KUKA KRL program: EPS_2_251806_MH01A_A_20260212042228.src

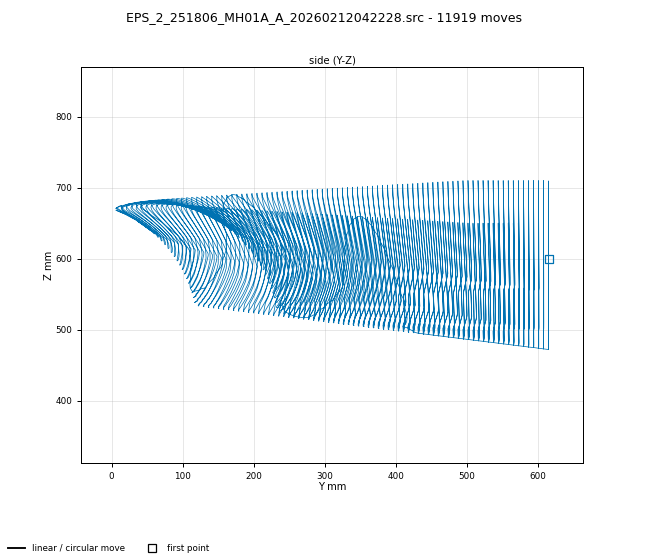
[picture p0: tool path of EPS_2_251806_MH01A_A_20260212042228.src, 11919 of 11921 moves have a stored position in this frame; points joined in program order, loops and branches not executed]
&ACCESS RVP
&REL 4
&COMMENT QRS 19112012
&PARAM EDITMASK = *
DEF PART()
EXT BAS (BAS_COMMAND :IN,REAL :IN )
INT I
BAS (#INITMOV,0 )

;KUKA QRS Post kuka4.cps  Date:22-06-2017 !

File_ID=3008

QRS_PRE_INIT()

;Init var - Until changes are made in qrs_pre_init
Outlet_Square_prg=0
Inlet_1_Square_prg=0
Inlet_2_Square_prg=0
Inlet_3_Square_prg=0
Inlet_4_Square_prg=0
Inlet_5_Square_prg=0

Outlet_1={X 0.000, Y 496.750, Z 561.000, B 0.000, E1 0.000 }
Inlet_1={X 0.000, Y 501.240, Z 501.000, B 0.000, E1 220.000 }
Outlet_1_type=299
Inlet_1_type=299
;QRS#1=Sidecore dimensions
;QRS#2=300-12" PVC SDR 35
;QRS#3=300-12" PVC SDR 35
;QRS#4=
;QRS#5=
;QRS#6=
;QRS#7=
;QRS#8=
;QRS#9=16M PSX
;QRS#10=16M PSX
;QRS#11=
;QRS#12=
;QRS#13=
;QRS#14=
;QRS#15=
;QRS#16=1220x127x991 3,25'
;QRS#17=EPS Height
;QRS#18=710,5
;QRS#19=*
;QRS#20= UPDATED VERSION 22-06-2017
;QRS#21=*
Outlet_Square=0150
Inlet_1_Square=0150
Inlet_2_Square=0
Inlet_3_Square=0
Inlet_4_Square=0
Inlet_5_Square=0
Mill_Square=1
Outlet_Square_Prg=206
Inlet_1_Square_prg=206

QRS_INIT()

$ADVANCE=5

; T1
PTP {E1 173.593,E2 173.593}
PTP {X 0,Y 615.505,A -85,B 0,C 180,E1 173.593,E2 173.593,E3 0,E4 0,E5 0,E6 0}
QRS_SPEED_INIT()
LIN {X 0,Y 615.505,Z 600,A -85,B 0,C 180,E1 173.593,E2 173.593,E3 0,E4 0,E5 0,E6 0} C_VEL
LIN {X 0,Y 615.505,Z 482.498,A -85,B 0,C 180,E1 173.593,E2 173.593} C_VEL
LIN {X 0,Y 615.505,Z 474.321,A -85,B 0,C 180,E1 173.593,E2 173.593} C_VEL
LIN {X 0,Y 615.491,Z 472.321,A -85,B 0,C 180,E1 173.407,E2 173.407} C_VEL
LIN {X 0,Y 615.481,Z 472.326,A -85,B 0,C 180,E1 170.801,E2 170.801} C_VEL
LIN {X 0,Y 615.48,Z 472.325,A -85,B 0,C 180,E1 168.139,E2 168.139} C_VEL
LIN {X 0,Y 615.489,Z 472.322,A -85,B 0,C 180,E1 165.451,E2 165.451} C_VEL
LIN {X 0,Y 615.493,Z 472.323,A -85,B 0,C 180,E1 162.729,E2 162.729} C_VEL
LIN {X 0,Y 615.484,Z 472.323,A -85,B 0,C 180,E1 159.967,E2 159.967} C_VEL
LIN {X 0,Y 615.483,Z 472.325,A -85,B 0,C 180,E1 157.155,E2 157.155} C_VEL
LIN {X 0,Y 615.498,Z 472.322,A -85,B 0,C 180,E1 154.284,E2 154.284} C_VEL
LIN {X 0,Y 615.484,Z 472.323,A -85,B 0,C 180,E1 151.548,E2 151.548} C_VEL
LIN {X 0,Y 615.482,Z 472.324,A -85,B 0,C 180,E1 148.912,E2 148.912} C_VEL
LIN {X 0,Y 615.491,Z 472.325,A -85,B 0,C 180,E1 146.463,E2 146.463} C_VEL
LIN {X 0,Y 615.483,Z 472.322,A -85,B 0,C 180,E1 143.574,E2 143.574} C_VEL
LIN {X 0,Y 615.495,Z 472.325,A -85,B 0,C 180,E1 140.935,E2 140.935} C_VEL
LIN {X 0,Y 615.496,Z 472.323,A -85,B 0,C 180,E1 138.526,E2 138.526} C_VEL
LIN {X 0,Y 615.482,Z 472.323,A -85,B 0,C 180,E1 135.849,E2 135.849} C_VEL
LIN {X 0,Y 615.486,Z 472.326,A -85,B 0,C 180,E1 133.047,E2 133.047} C_VEL
LIN {X 0,Y 615.496,Z 472.322,A -85,B 0,C 180,E1 130.089,E2 130.089} C_VEL
LIN {X 0,Y 615.491,Z 472.321,A -85,B 0,C 180,E1 127.241,E2 127.241} C_VEL
LIN {X 0,Y 615.483,Z 472.323,A -85,B 0,C 180,E1 124.699,E2 124.699} C_VEL
LIN {X 0,Y 615.487,Z 472.325,A -85,B 0,C 180,E1 122.33,E2 122.33} C_VEL
LIN {X 0,Y 615.486,Z 472.325,A -85,B 0,C 180,E1 119.793,E2 119.793} C_VEL
LIN {X 0,Y 615.491,Z 472.321,A -85,B 0,C 180,E1 117.045,E2 117.045} C_VEL
LIN {X 0,Y 615.497,Z 472.322,A -85,B 0,C 180,E1 114.271,E2 114.271} C_VEL
LIN {X 0,Y 615.48,Z 472.325,A -85,B 0,C 180,E1 111.431,E2 111.431} C_VEL
LIN {X 0,Y 615.484,Z 472.323,A -85,B 0,C 180,E1 108.602,E2 108.602} C_VEL
LIN {X 0,Y 615.495,Z 472.321,A -85,B 0,C 180,E1 105.904,E2 105.904} C_VEL
LIN {X 0,Y 615.487,Z 472.324,A -85,B 0,C 180,E1 103.201,E2 103.201} C_VEL
LIN {X 0,Y 615.48,Z 472.324,A -85,B 0,C 180,E1 100.527,E2 100.527} C_VEL
LIN {X 0,Y 615.489,Z 472.326,A -85,B 0,C 180,E1 97.875,E2 97.875} C_VEL
LIN {X 0,Y 615.484,Z 472.322,A -85,B 0,C 180,E1 95.241,E2 95.241} C_VEL
LIN {X 0,Y 615.483,Z 472.325,A -85,B 0,C 180,E1 92.617,E2 92.617} C_VEL
LIN {X 0,Y 615.492,Z 472.323,A -85,B 0,C 180,E1 90,E2 90} C_VEL
LIN {X 0,Y 615.498,Z 472.416,A -85,B 0,C 180,E1 88.037,E2 88.037} C_VEL
LIN {X 0,Y 615.48,Z 475.112,A -85,B 0,C 180,E1 85.415,E2 85.415} C_VEL
LIN {X 0,Y 615.489,Z 477.991,A -85,B 0,C 180,E1 82.784,E2 82.784} C_VEL
LIN {X 0,Y 615.484,Z 480.998,A -85,B 0,C 180,E1 80.138,E2 80.138} C_VEL
LIN {X 0,Y 615.491,Z 484.127,A -85,B 0,C 180,E1 77.47,E2 77.47} C_VEL
LIN {X 0,Y 615.489,Z 487.344,A -85,B 0,C 180,E1 74.774,E2 74.774} C_VEL
LIN {X 0,Y 615.487,Z 490.698,A -85,B 0,C 180,E1 72.043,E2 72.043} C_VEL
LIN {X 0,Y 615.478,Z 494.15,A -85,B 0,C 180,E1 69.269,E2 69.269} C_VEL
LIN {X 0,Y 615.48,Z 496.826,A -85,B 0,C 180,E1 67.155,E2 67.155} C_VEL
LIN {X 0,Y 615.477,Z 498.079,A -85,B 0,C 180,E1 66.288,E2 66.288} C_VEL
LIN {X 0,Y 615.487,Z 512.595,A -85,B 0,C 180,E1 66.049,E2 66.049} C_VEL
LIN {X 0,Y 615.485,Z 527.058,A -85,B 0,C 180,E1 65.683,E2 65.683} C_VEL
LIN {X 0,Y 615.479,Z 541.48,A -85,B 0,C 180,E1 65.188,E2 65.188} C_VEL
LIN {X 0,Y 615.481,Z 555.329,A -85,B 0,C 180,E1 64.578,E2 64.578} C_VEL
LIN {X 0,Y 615.499,Z 568.988,A -85,B 0,C 180,E1 63.83,E2 63.83} C_VEL
LIN {X 0,Y 615.498,Z 582.101,A -85,B 0,C 180,E1 62.954,E2 62.954} C_VEL
LIN {X 0,Y 615.493,Z 592.977,A -85,B 0,C 180,E1 62.085,E2 62.085} C_VEL
LIN {X 0,Y 615.494,Z 602.897,A -85,B 0,C 180,E1 61.156,E2 61.156} C_VEL
LIN {X 0,Y 615.497,Z 613.099,A -85,B 0,C 180,E1 60.023,E2 60.023} C_VEL
LIN {X 0,Y 615.497,Z 622.489,A -85,B 0,C 180,E1 58.765,E2 58.765} C_VEL
LIN {X 0,Y 615.493,Z 629.992,A -85,B 0,C 180,E1 57.543,E2 57.543} C_VEL
LIN {X 0,Y 615.492,Z 636.558,A -85,B 0,C 180,E1 56.223,E2 56.223} C_VEL
LIN {X 0,Y 615.487,Z 640.708,A -85,B 0,C 180,E1 55.185,E2 55.185} C_VEL
LIN {X 0,Y 615.493,Z 643.983,A -85,B 0,C 180,E1 54.166,E2 54.166} C_VEL
LIN {X 0,Y 615.493,Z 647.292,A -85,B 0,C 180,E1 52.759,E2 52.759} C_VEL
LIN {X 0,Y 615.494,Z 648.577,A -85,B 0,C 180,E1 51.932,E2 51.932} C_VEL
LIN {X 0,Y 615.49,Z 649.536,A -85,B 0,C 180,E1 50.938,E2 50.938} C_VEL
LIN {X 0,Y 615.498,Z 649.883,A -85,B 0,C 180,E1 49.91,E2 49.91} C_VEL
LIN {X 0,Y 615.491,Z 649.22,A -85,B 0,C 180,E1 48.527,E2 48.527} C_VEL
LIN {X 0,Y 615.491,Z 646.908,A -85,B 0,C 180,E1 46.953,E2 46.953} C_VEL
LIN {X 0,Y 615.493,Z 643.151,A -85,B 0,C 180,E1 45.461,E2 45.461} C_VEL
LIN {X 0,Y 615.492,Z 638.543,A -85,B 0,C 180,E1 44.15,E2 44.15} C_VEL
LIN {X 0,Y 615.494,Z 631.812,A -85,B 0,C 180,E1 42.7,E2 42.7} C_VEL
LIN {X 0,Y 615.495,Z 624.699,A -85,B 0,C 180,E1 41.474,E2 41.474} C_VEL
LIN {X 0,Y 615.496,Z 615.806,A -85,B 0,C 180,E1 40.22,E2 40.22} C_VEL
LIN {X 0,Y 615.495,Z 605.907,A -85,B 0,C 180,E1 39.064,E2 39.064} C_VEL
LIN {X 0,Y 615.496,Z 595.163,A -85,B 0,C 180,E1 38.014,E2 38.014} C_VEL
LIN {X 0,Y 615.495,Z 582.905,A -85,B 0,C 180,E1 37.014,E2 37.014} C_VEL
LIN {X 0,Y 615.497,Z 569.826,A -85,B 0,C 180,E1 36.13,E2 36.13} C_VEL
LIN {X 0,Y 615.481,Z 556.024,A -85,B 0,C 180,E1 35.366,E2 35.366} C_VEL
LIN {X 0,Y 615.49,Z 542.45,A -85,B 0,C 180,E1 34.759,E2 34.759} C_VEL
LIN {X 0,Y 615.477,Z 527.351,A -85,B 0,C 180,E1 34.235,E2 34.235} C_VEL
LIN {X 0,Y 615.487,Z 513.002,A -85,B 0,C 180,E1 33.87,E2 33.87} C_VEL
LIN {X 0,Y 615.491,Z 497.929,A -85,B 0,C 180,E1 33.611,E2 33.611} C_VEL
LIN {X 0,Y 615.483,Z 494.501,A -85,B 0,C 180,E1 30.92,E2 30.92} C_VEL
LIN {X 0,Y 615.483,Z 491.414,A -85,B 0,C 180,E1 28.451,E2 28.451} C_VEL
LIN {X 0,Y 615.493,Z 487.874,A -85,B 0,C 180,E1 25.571,E2 25.571} C_VEL
LIN {X 0,Y 615.482,Z 484.601,A -85,B 0,C 180,E1 22.845,E2 22.845} C_VEL
LIN {X 0,Y 615.477,Z 481.304,A -85,B 0,C 180,E1 20.033,E2 20.033} C_VEL
LIN {X 0,Y 615.492,Z 478.15,A -85,B 0,C 180,E1 17.271,E2 17.271} C_VEL
LIN {X 0,Y 615.487,Z 475.186,A -85,B 0,C 180,E1 14.549,E2 14.549} C_VEL
LIN {X 0,Y 615.485,Z 472.509,A -85,B 0,C 180,E1 11.861,E2 11.861} C_VEL
LIN {X 0,Y 615.479,Z 472.312,A -85,B 0,C 180,E1 9.199,E2 9.199} C_VEL
LIN {X 0,Y 615.491,Z 472.313,A -85,B 0,C 180,E1 6.557,E2 6.557} C_VEL
LIN {X 0,Y 615.488,Z 472.319,A -85,B 0,C 180,E1 3.929,E2 3.929} C_VEL
LIN {X 0,Y 615.485,Z 472.309,A -85,B 0,C 180,E1 1.309,E2 1.309} C_VEL
LIN {X 0,Y 615.485,Z 472.321,A -85,B 0,C 180,E1 -1.308,E2 -1.308} C_VEL
LIN {X 0,Y 615.475,Z 472.316,A -85,B 0,C 180,E1 -3.928,E2 -3.928} C_VEL
LIN {X 0,Y 615.492,Z 472.31,A -85,B 0,C 180,E1 -6.588,E2 -6.588} C_VEL
LIN {X 0,Y 615.487,Z 472.325,A -85,B 0,C 180,E1 -9.199,E2 -9.199} C_VEL
LIN {X 0,Y 615.479,Z 472.311,A -85,B 0,C 180,E1 -11.861,E2 -11.861} C_VEL
LIN {X 0,Y 615.491,Z 472.318,A -85,B 0,C 180,E1 -14.549,E2 -14.549} C_VEL
LIN {X 0,Y 615.48,Z 472.314,A -85,B 0,C 180,E1 -17.271,E2 -17.271} C_VEL
LIN {X 0,Y 615.479,Z 472.316,A -85,B 0,C 180,E1 -20.033,E2 -20.033} C_VEL
LIN {X 0,Y 615.482,Z 472.316,A -85,B 0,C 180,E1 -22.845,E2 -22.845} C_VEL
LIN {X 0,Y 615.493,Z 472.312,A -85,B 0,C 180,E1 -25.715,E2 -25.715} C_VEL
LIN {X 0,Y 615.489,Z 472.312,A -85,B 0,C 180,E1 -28.658,E2 -28.658} C_VEL
LIN {X 0,Y 615.477,Z 472.312,A -85,B 0,C 180,E1 -31.085,E2 -31.085} C_VEL
LIN {X 0,Y 615.485,Z 472.319,A -85,B 0,C 180,E1 -33.535,E2 -33.535} C_VEL
LIN {X 0,Y 615.486,Z 472.323,A -85,B 0,C 180,E1 -35.834,E2 -35.834} C_VEL
LIN {X 0,Y 615.478,Z 472.316,A -85,B 0,C 180,E1 -38.069,E2 -38.069} C_VEL
LIN {X 0,Y 615.484,Z 472.31,A -85,B 0,C 180,E1 -40.607,E2 -40.607} C_VEL
LIN {X 0,Y 615.497,Z 472.324,A -85,B 0,C 180,E1 -43.244,E2 -43.244} C_VEL
LIN {X 0,Y 615.482,Z 472.31,A -85,B 0,C 180,E1 -46.003,E2 -46.003} C_VEL
LIN {X 0,Y 615.492,Z 472.352,A -85,B 0,C 180,E1 -48.716,E2 -48.716} C_VEL
LIN {X 0,Y 615.483,Z 479.207,A -85,B 0,C 180,E1 -51.096,E2 -51.096} C_VEL
LIN {X 0,Y 615.486,Z 486.794,A -85,B 0,C 180,E1 -53.576,E2 -53.576} C_VEL
LIN {X 0,Y 615.496,Z 495.763,A -85,B 0,C 180,E1 -56.465,E2 -56.465} C_VEL
LIN {X 0,Y 615.478,Z 504.122,A -85,B 0,C 180,E1 -59.08,E2 -59.08} C_VEL
LIN {X 0,Y 615.481,Z 512.228,A -85,B 0,C 180,E1 -61.551,E2 -61.551} C_VEL
LIN {X 0,Y 615.493,Z 521.4,A -85,B 0,C 180,E1 -64.285,E2 -64.285} C_VEL
LIN {X 0,Y 615.48,Z 531.274,A -85,B 0,C 180,E1 -67.155,E2 -67.155} C_VEL
LIN {X 0,Y 615.492,Z 541.126,A -85,B 0,C 180,E1 -69.967,E2 -69.967} C_VEL
LIN {X 0,Y 615.485,Z 550.985,A -85,B 0,C 180,E1 -72.729,E2 -72.729} C_VEL
LIN {X 0,Y 615.489,Z 554.183,A -85,B 0,C 180,E1 -73.618,E2 -73.618} C_VEL
LIN {X 0,Y 615.495,Z 570.381,A -85,B 0,C 180,E1 -73.865,E2 -73.865} C_VEL
LIN {X 0,Y 615.48,Z 585.284,A -85,B 0,C 180,E1 -74.222,E2 -74.222} C_VEL
LIN {X 0,Y 615.484,Z 599.424,A -85,B 0,C 180,E1 -74.689,E2 -74.689} C_VEL
LIN {X 0,Y 615.485,Z 613.357,A -85,B 0,C 180,E1 -75.282,E2 -75.282} C_VEL
LIN {X 0,Y 615.499,Z 626.673,A -85,B 0,C 180,E1 -75.986,E2 -75.986} C_VEL
LIN {X 0,Y 615.498,Z 639.314,A -85,B 0,C 180,E1 -76.799,E2 -76.799} C_VEL
LIN {X 0,Y 615.496,Z 650.292,A -85,B 0,C 180,E1 -77.637,E2 -77.637} C_VEL
LIN {X 0,Y 615.497,Z 661.353,A -85,B 0,C 180,E1 -78.64,E2 -78.64} C_VEL
LIN {X 0,Y 615.496,Z 672.068,A -85,B 0,C 180,E1 -79.806,E2 -79.806} C_VEL
LIN {X 0,Y 615.497,Z 680.987,A -85,B 0,C 180,E1 -80.967,E2 -80.967} C_VEL
LIN {X 0,Y 615.494,Z 688.391,A -85,B 0,C 180,E1 -82.124,E2 -82.124} C_VEL
LIN {X 0,Y 615.49,Z 695.271,A -85,B 0,C 180,E1 -83.443,E2 -83.443} C_VEL
LIN {X 0,Y 615.491,Z 700.665,A -85,B 0,C 180,E1 -84.759,E2 -84.759} C_VEL
LIN {X 0,Y 615.495,Z 704.739,A -85,B 0,C 180,E1 -86.071,E2 -86.071} C_VEL
LIN {X 0,Y 615.495,Z 707.599,A -85,B 0,C 180,E1 -87.382,E2 -87.382} C_VEL
LIN {X 0,Y 615.493,Z 709.306,A -85,B 0,C 180,E1 -88.691,E2 -88.691} C_VEL
LIN {X 0,Y 615.491,Z 709.889,A -85,B 0,C 180,E1 -90,E2 -90} C_VEL
LIN {X 0,Y 615.493,Z 709.307,A -85,B 0,C 180,E1 -91.308,E2 -91.308} C_VEL
LIN {X 0,Y 615.495,Z 707.6,A -85,B 0,C 180,E1 -92.617,E2 -92.617} C_VEL
LIN {X 0,Y 615.495,Z 704.741,A -85,B 0,C 180,E1 -93.928,E2 -93.928} C_VEL
LIN {X 0,Y 615.491,Z 700.668,A -85,B 0,C 180,E1 -95.241,E2 -95.241} C_VEL
LIN {X 0,Y 615.49,Z 695.155,A -85,B 0,C 180,E1 -96.581,E2 -96.581} C_VEL
LIN {X 0,Y 615.494,Z 688.396,A -85,B 0,C 180,E1 -97.875,E2 -97.875} C_VEL
LIN {X 0,Y 615.497,Z 679.812,A -85,B 0,C 180,E1 -99.198,E2 -99.198} C_VEL
LIN {X 0,Y 615.494,Z 670.672,A -85,B 0,C 180,E1 -100.36,E2 -100.36} C_VEL
LIN {X 0,Y 615.497,Z 661.359,A -85,B 0,C 180,E1 -101.359,E2 -101.359} C_VEL
LIN {X 0,Y 615.496,Z 650.3,A -85,B 0,C 180,E1 -102.362,E2 -102.362} C_VEL
LIN {X 0,Y 615.498,Z 638.161,A -85,B 0,C 180,E1 -103.284,E2 -103.284} C_VEL
LIN {X 0,Y 615.498,Z 625.407,A -85,B 0,C 180,E1 -104.089,E2 -104.089} C_VEL
LIN {X 0,Y 615.486,Z 611.623,A -85,B 0,C 180,E1 -104.802,E2 -104.802} C_VEL
LIN {X 0,Y 615.48,Z 597.199,A -85,B 0,C 180,E1 -105.395,E2 -105.395} C_VEL
LIN {X 0,Y 615.484,Z 582.272,A -85,B 0,C 180,E1 -105.862,E2 -105.862} C_VEL
LIN {X 0,Y 615.496,Z 566.874,A -85,B 0,C 180,E1 -106.2,E2 -106.2} C_VEL
LIN {X 0,Y 615.489,Z 554.125,A -85,B 0,C 180,E1 -106.398,E2 -106.398} C_VEL
LIN {X 0,Y 615.485,Z 544.833,A -85,B 0,C 180,E1 -108.991,E2 -108.991} C_VEL
LIN {X 0,Y 615.486,Z 534.967,A -85,B 0,C 180,E1 -111.783,E2 -111.783} C_VEL
LIN {X 0,Y 615.487,Z 526.34,A -85,B 0,C 180,E1 -114.271,E2 -114.271} C_VEL
LIN {X 0,Y 615.491,Z 516.906,A -85,B 0,C 180,E1 -117.046,E2 -117.046} C_VEL
LIN {X 0,Y 615.485,Z 507.787,A -85,B 0,C 180,E1 -119.794,E2 -119.794} C_VEL
LIN {X 0,Y 615.481,Z 499.186,A -85,B 0,C 180,E1 -122.457,E2 -122.457} C_VEL
LIN {X 0,Y 615.496,Z 490.532,A -85,B 0,C 180,E1 -125.213,E2 -125.213} C_VEL
LIN {X 0,Y 615.489,Z 481.785,A -85,B 0,C 180,E1 -128.067,E2 -128.067} C_VEL
LIN {X 0,Y 615.477,Z 474.341,A -85,B 0,C 180,E1 -130.606,E2 -130.606} C_VEL
LIN {X 0,Y 615.49,Z 472.322,A -85,B 0,C 180,E1 -131.378,E2 -131.378} C_VEL
LIN {X 0,Y 615.492,Z 472.323,A -85,B 0,C 180,E1 -134.148,E2 -134.148} C_VEL
LIN {X 0,Y 615.488,Z 472.322,A -85,B 0,C 180,E1 -136.951,E2 -136.951} C_VEL
LIN {X 0,Y 615.495,Z 472.325,A -85,B 0,C 180,E1 -139.908,E2 -139.908} C_VEL
LIN {X 0,Y 615.481,Z 472.324,A -85,B 0,C 180,E1 -142.758,E2 -142.758} C_VEL
LIN {X 0,Y 615.491,Z 472.326,A -85,B 0,C 180,E1 -145.297,E2 -145.297} C_VEL
LIN {X 0,Y 615.49,Z 472.325,A -85,B 0,C 180,E1 -147.667,E2 -147.667} C_VEL
LIN {X 0,Y 615.488,Z 472.322,A -85,B 0,C 180,E1 -150.203,E2 -150.203} C_VEL
LIN {X 0,Y 615.492,Z 472.325,A -85,B 0,C 180,E1 -152.951,E2 -152.951} C_VEL
LIN {X 0,Y 615.479,Z 472.323,A -85,B 0,C 180,E1 -155.728,E2 -155.728} C_VEL
LIN {X 0,Y 615.499,Z 472.325,A -85,B 0,C 180,E1 -158.569,E2 -158.569} C_VEL
LIN {X 0,Y 615.495,Z 472.32,A -85,B 0,C 180,E1 -161.389,E2 -161.389} C_VEL
LIN {X 0,Y 615.491,Z 472.326,A -85,B 0,C 180,E1 -164.095,E2 -164.095} C_VEL
LIN {X 0,Y 615.48,Z 472.323,A -85,B 0,C 180,E1 -166.799,E2 -166.799} C_VEL
LIN {X 0,Y 615.495,Z 472.324,A -85,B 0,C 180,E1 -169.473,E2 -169.473} C_VEL
LIN {X 0,Y 615.483,Z 472.323,A -85,B 0,C 180,E1 -172.125,E2 -172.125} C_VEL
LIN {X 0,Y 615.487,Z 472.323,A -85,B 0,C 180,E1 -174.759,E2 -174.759} C_VEL
LIN {X 0,Y 615.496,Z 472.324,A -85,B 0,C 180,E1 -177.382,E2 -177.382} C_VEL
LIN {X 0,Y 615.477,Z 472.324,A -85,B 0,C 180,E1 -180,E2 -180} C_VEL
LIN {X 0,Y 615.494,Z 472.323,A -85,B 0,C 180,E1 -182.618,E2 -182.618} C_VEL
LIN {X 0,Y 615.491,Z 472.323,A -85,B 0,C 180,E1 -185.241,E2 -185.241} C_VEL
LIN {X 0,Y 615.491,Z 472.321,A -85,B 0,C 180,E1 -186.593,E2 -186.593} C_VEL
LIN {X 0,Y 614.815,Z 472.47,A -85,B 0,C 180,E1 -187.139,E2 -187.139} C_VEL
LIN {X 0,Y 611.975,Z 472.882,A -85,B 0,C 180,E1 -188.025,E2 -188.025} C_VEL
LIN {X 0,Y 609.579,Z 473.194,A -85,B 0,C 180,E1 -188.737,E2 -188.737} C_VEL
LIN {X 0,Y 608.542,Z 473.312,A -85,B 0,C 180,E1 -189.287,E2 -189.287} C_VEL
LIN {X 0,Y 608.453,Z 473.321,A -85,B 0,C 180,E1 -189.473,E2 -189.473} C_VEL
LIN {X 0,Y 608.457,Z 473.32,A -85,B 0,C 180,E1 -192,E2 -192} C_VEL
LIN {X 0,Y 608.476,Z 473.319,A -85,B 0,C 180,E1 -194.721,E2 -194.721} C_VEL
LIN {X 0,Y 608.457,Z 473.32,A -85,B 0,C 180,E1 -197.477,E2 -197.477} C_VEL
LIN {X 0,Y 608.462,Z 473.321,A -85,B 0,C 180,E1 -200.275,E2 -200.275} C_VEL
LIN {X 0,Y 608.449,Z 473.322,A -85,B 0,C 180,E1 -202.477,E2 -202.477} C_VEL
LIN {X 0,Y 608.453,Z 473.32,A -85,B 0,C 180,E1 -205.301,E2 -205.301} C_VEL
LIN {X 0,Y 608.454,Z 473.32,A -85,B 0,C 180,E1 -207.518,E2 -207.518} C_VEL
LIN {X 0,Y 608.471,Z 473.318,A -85,B 0,C 180,E1 -209.975,E2 -209.975} C_VEL
LIN {X 0,Y 608.465,Z 473.322,A -85,B 0,C 180,E1 -212.525,E2 -212.525} C_VEL
LIN {X 0,Y 608.449,Z 473.32,A -85,B 0,C 180,E1 -215.278,E2 -215.278} C_VEL
LIN {X 0,Y 608.471,Z 473.319,A -85,B 0,C 180,E1 -217.747,E2 -217.747} C_VEL
LIN {X 0,Y 608.477,Z 473.319,A -85,B 0,C 180,E1 -220.334,E2 -220.334} C_VEL
LIN {X 0,Y 608.471,Z 473.319,A -85,B 0,C 180,E1 -223.31,E2 -223.31} C_VEL
LIN {X 0,Y 608.469,Z 473.318,A -85,B 0,C 180,E1 -226.132,E2 -226.132} C_VEL
LIN {X 0,Y 608.461,Z 473.32,A -85,B 0,C 180,E1 -228.825,E2 -228.825} C_VEL
LIN {X 0,Y 608.473,Z 473.317,A -85,B 0,C 180,E1 -231.76,E2 -231.76} C_VEL
LIN {X 0,Y 608.478,Z 473.317,A -85,B 0,C 180,E1 -233.951,E2 -233.951} C_VEL
LIN {X 0,Y 608.463,Z 473.319,A -85,B 0,C 180,E1 -236.33,E2 -236.33} C_VEL
LIN {X 0,Y 608.479,Z 473.318,A -85,B 0,C 180,E1 -238.728,E2 -238.728} C_VEL
LIN {X 0,Y 608.477,Z 473.318,A -85,B 0,C 180,E1 -241.38,E2 -241.38} C_VEL
LIN {X 0,Y 608.479,Z 473.318,A -85,B 0,C 180,E1 -244.279,E2 -244.279} C_VEL
LIN {X 0,Y 608.45,Z 473.321,A -85,B 0,C 180,E1 -246.877,E2 -246.877} C_VEL
LIN {X 0,Y 608.461,Z 473.319,A -85,B 0,C 180,E1 -249.324,E2 -249.324} C_VEL
LIN {X 0,Y 608.455,Z 473.32,A -85,B 0,C 180,E1 -251.829,E2 -251.829} C_VEL
LIN {X 0,Y 608.476,Z 473.318,A -85,B 0,C 180,E1 -254.595,E2 -254.595} C_VEL
LIN {X 0,Y 608.473,Z 473.318,A -85,B 0,C 180,E1 -257.324,E2 -257.324} C_VEL
LIN {X 0,Y 608.454,Z 473.321,A -85,B 0,C 180,E1 -260.023,E2 -260.023} C_VEL
LIN {X 0,Y 608.467,Z 473.318,A -85,B 0,C 180,E1 -262.701,E2 -262.701} C_VEL
LIN {X 0,Y 608.463,Z 473.322,A -85,B 0,C 180,E1 -265.363,E2 -265.363} C_VEL
LIN {X 0,Y 608.466,Z 473.318,A -85,B 0,C 180,E1 -268.015,E2 -268.015} C_VEL
LIN {X 0,Y 608.481,Z 473.318,A -85,B 0,C 180,E1 -270.662,E2 -270.662} C_VEL
LIN {X 0,Y 608.465,Z 473.322,A -85,B 0,C 180,E1 -271.986,E2 -271.986} C_VEL
LIN {X 0,Y 608.449,Z 476,A -85,B 0,C 180,E1 -274.638,E2 -274.638} C_VEL
LIN {X 0,Y 608.453,Z 478.867,A -85,B 0,C 180,E1 -277.3,E2 -277.3} C_VEL
LIN {X 0,Y 608.421,Z 481.906,A -85,B 0,C 180,E1 -279.978,E2 -279.978} C_VEL
LIN {X 0,Y 608.423,Z 485.051,A -85,B 0,C 180,E1 -282.678,E2 -282.678} C_VEL
LIN {X 0,Y 608.419,Z 488.309,A -85,B 0,C 180,E1 -285.407,E2 -285.407} C_VEL
LIN {X 0,Y 608.411,Z 491.684,A -85,B 0,C 180,E1 -288.173,E2 -288.173} C_VEL
LIN {X 0,Y 608.413,Z 495.181,A -85,B 0,C 180,E1 -290.983,E2 -290.983} C_VEL
LIN {X 0,Y 608.429,Z 498.373,A -85,B 0,C 180,E1 -293.508,E2 -293.508} C_VEL
LIN {X 0,Y 608.664,Z 502.587,A -85,B 0,C 180,E1 -293.588,E2 -293.588} C_VEL
LIN {X 0,Y 608.664,Z 517.473,A -85,B 0,C 180,E1 -293.879,E2 -293.879} C_VEL
LIN {X 0,Y 608.622,Z 532.678,A -85,B 0,C 180,E1 -294.315,E2 -294.315} C_VEL
LIN {X 0,Y 608.612,Z 547.393,A -85,B 0,C 180,E1 -294.883,E2 -294.883} C_VEL
LIN {X 0,Y 608.566,Z 561.722,A -85,B 0,C 180,E1 -295.586,E2 -295.586} C_VEL
LIN {X 0,Y 608.539,Z 575.136,A -85,B 0,C 180,E1 -296.4,E2 -296.4} C_VEL
LIN {X 0,Y 608.528,Z 587.703,A -85,B 0,C 180,E1 -297.323,E2 -297.323} C_VEL
LIN {X 0,Y 608.485,Z 598.497,A -85,B 0,C 180,E1 -298.265,E2 -298.265} C_VEL
LIN {X 0,Y 608.484,Z 609.409,A -85,B 0,C 180,E1 -299.398,E2 -299.398} C_VEL
LIN {X 0,Y 608.454,Z 618.664,A -85,B 0,C 180,E1 -300.545,E2 -300.545} C_VEL
LIN {X 0,Y 608.46,Z 626.494,A -85,B 0,C 180,E1 -301.705,E2 -301.705} C_VEL
LIN {X 0,Y 608.442,Z 633.124,A -85,B 0,C 180,E1 -302.88,E2 -302.88} C_VEL
LIN {X 0,Y 608.44,Z 638.578,A -85,B 0,C 180,E1 -304.071,E2 -304.071} C_VEL
LIN {X 0,Y 608.424,Z 642.973,A -85,B 0,C 180,E1 -305.279,E2 -305.279} C_VEL
LIN {X 0,Y 608.422,Z 645.348,A -85,B 0,C 180,E1 -306.094,E2 -306.094} C_VEL
LIN {X 0,Y 608.431,Z 647.777,A -85,B 0,C 180,E1 -307.153,E2 -307.153} C_VEL
LIN {X 0,Y 608.413,Z 649.814,A -85,B 0,C 180,E1 -308.592,E2 -308.592} C_VEL
LIN {X 0,Y 608.412,Z 650.365,A -85,B 0,C 180,E1 -309.444,E2 -309.444} C_VEL
LIN {X 0,Y 608.433,Z 650.44,A -85,B 0,C 180,E1 -310.326,E2 -310.326} C_VEL
LIN {X 0,Y 608.415,Z 649.935,A -85,B 0,C 180,E1 -311.337,E2 -311.337} C_VEL
LIN {X 0,Y 608.437,Z 648.787,A -85,B 0,C 180,E1 -312.331,E2 -312.331} C_VEL
LIN {X 0,Y 608.436,Z 646.996,A -85,B 0,C 180,E1 -313.305,E2 -313.305} C_VEL
LIN {X 0,Y 608.423,Z 643.014,A -85,B 0,C 180,E1 -314.798,E2 -314.798} C_VEL
LIN {X 0,Y 608.429,Z 638.119,A -85,B 0,C 180,E1 -316.126,E2 -316.126} C_VEL
LIN {X 0,Y 608.44,Z 632.234,A -85,B 0,C 180,E1 -317.38,E2 -317.38} C_VEL
LIN {X 0,Y 608.443,Z 624.802,A -85,B 0,C 180,E1 -318.659,E2 -318.659} C_VEL
LIN {X 0,Y 608.474,Z 615.89,A -85,B 0,C 180,E1 -319.914,E2 -319.914} C_VEL
LIN {X 0,Y 608.494,Z 606.137,A -85,B 0,C 180,E1 -321.058,E2 -321.058} C_VEL
LIN {X 0,Y 608.497,Z 595.228,A -85,B 0,C 180,E1 -322.13,E2 -322.13} C_VEL
LIN {X 0,Y 608.518,Z 583.622,A -85,B 0,C 180,E1 -323.089,E2 -323.089} C_VEL
LIN {X 0,Y 608.548,Z 571.35,A -85,B 0,C 180,E1 -323.941,E2 -323.941} C_VEL
LIN {X 0,Y 608.576,Z 557.516,A -85,B 0,C 180,E1 -324.731,E2 -324.731} C_VEL
LIN {X 0,Y 608.624,Z 543.685,A -85,B 0,C 180,E1 -325.368,E2 -325.368} C_VEL
LIN {X 0,Y 608.633,Z 528.133,A -85,B 0,C 180,E1 -325.924,E2 -325.924} C_VEL
LIN {X 0,Y 608.675,Z 512.3,A -85,B 0,C 180,E1 -326.329,E2 -326.329} C_VEL
LIN {X 0,Y 608.519,Z 499.111,A -85,B 0,C 180,E1 -326.556,E2 -326.556} C_VEL
LIN {X 0,Y 608.415,Z 498.384,A -85,B 0,C 180,E1 -326.574,E2 -326.574} C_VEL
LIN {X 0,Y 608.422,Z 494.748,A -85,B 0,C 180,E1 -329.452,E2 -329.452} C_VEL
LIN {X 0,Y 608.431,Z 491.912,A -85,B 0,C 180,E1 -331.732,E2 -331.732} C_VEL
LIN {X 0,Y 608.43,Z 488.29,A -85,B 0,C 180,E1 -334.698,E2 -334.698} C_VEL
LIN {X 0,Y 608.428,Z 484.838,A -85,B 0,C 180,E1 -337.593,E2 -337.593} C_VEL
LIN {X 0,Y 608.43,Z 481.542,A -85,B 0,C 180,E1 -340.428,E2 -340.428} C_VEL
LIN {X 0,Y 608.447,Z 478.394,A -85,B 0,C 180,E1 -343.215,E2 -343.215} C_VEL
LIN {X 0,Y 608.454,Z 475.497,A -85,B 0,C 180,E1 -345.986,E2 -345.986} C_VEL
LIN {X 0,Y 608.445,Z 473.518,A -85,B 0,C 180,E1 -348,E2 -348} C_VEL
LIN {X 0,Y 608.465,Z 473.32,A -85,B 0,C 180,E1 -350.023,E2 -350.023} C_VEL
LIN {X 0,Y 608.46,Z 473.313,A -85,B 0,C 180,E1 -352.7,E2 -352.7} C_VEL
LIN {X 0,Y 608.462,Z 473.315,A -85,B 0,C 180,E1 -355.362,E2 -355.362} C_VEL
LIN {X 0,Y 608.457,Z 473.318,A -85,B 0,C 180,E1 -358.014,E2 -358.014} C_VEL
LIN {X 0,Y 608.479,Z 473.31,A -85,B 0,C 180,E1 -360.662,E2 -360.662} C_VEL
LIN {X 0,Y 608.476,Z 473.318,A -85,B 0,C 180,E1 -363.31,E2 -363.31} C_VEL
LIN {X 0,Y 608.454,Z 473.314,A -85,B 0,C 180,E1 -365.967,E2 -365.967} C_VEL
LIN {X 0,Y 608.46,Z 473.315,A -85,B 0,C 180,E1 -368.636,E2 -368.636} C_VEL
LIN {X 0,Y 608.471,Z 473.316,A -85,B 0,C 180,E1 -371.324,E2 -371.324} C_VEL
LIN {X 0,Y 608.463,Z 473.312,A -85,B 0,C 180,E1 -374.037,E2 -374.037} C_VEL
LIN {X 0,Y 608.475,Z 473.319,A -85,B 0,C 180,E1 -376.783,E2 -376.783} C_VEL
LIN {X 0,Y 608.447,Z 473.314,A -85,B 0,C 180,E1 -379.571,E2 -379.571} C_VEL
LIN {X 0,Y 608.471,Z 473.321,A -85,B 0,C 180,E1 -382.405,E2 -382.405} C_VEL
LIN {X 0,Y 608.451,Z 473.319,A -85,B 0,C 180,E1 -384.571,E2 -384.571} C_VEL
LIN {X 0,Y 608.471,Z 473.311,A -85,B 0,C 180,E1 -387.207,E2 -387.207} C_VEL
LIN {X 0,Y 608.47,Z 473.321,A -85,B 0,C 180,E1 -389.973,E2 -389.973} C_VEL
LIN {X 0,Y 608.462,Z 473.313,A -85,B 0,C 180,E1 -392.523,E2 -392.523} C_VEL
LIN {X 0,Y 608.449,Z 473.317,A -85,B 0,C 180,E1 -395.277,E2 -395.277} C_VEL
LIN {X 0,Y 608.464,Z 473.319,A -85,B 0,C 180,E1 -397.746,E2 -397.746} C_VEL
LIN {X 0,Y 608.446,Z 473.314,A -85,B 0,C 180,E1 -400.329,E2 -400.329} C_VEL
LIN {X 0,Y 608.482,Z 473.32,A -85,B 0,C 180,E1 -403.311,E2 -403.311} C_VEL
LIN {X 0,Y 608.469,Z 473.312,A -85,B 0,C 180,E1 -406.131,E2 -406.131} C_VEL
LIN {X 0,Y 608.476,Z 473.373,A -85,B 0,C 180,E1 -408.522,E2 -408.522} C_VEL
LIN {X 0,Y 608.543,Z 479.468,A -85,B 0,C 180,E1 -410.694,E2 -410.694} C_VEL
LIN {X 0,Y 608.518,Z 487.918,A -85,B 0,C 180,E1 -413.503,E2 -413.503} C_VEL
LIN {X 0,Y 608.525,Z 495.494,A -85,B 0,C 180,E1 -415.934,E2 -415.934} C_VEL
LIN {X 0,Y 608.521,Z 504.27,A -85,B 0,C 180,E1 -418.721,E2 -418.721} C_VEL
LIN {X 0,Y 608.493,Z 512.881,A -85,B 0,C 180,E1 -421.376,E2 -421.376} C_VEL
LIN {X 0,Y 608.496,Z 522.524,A -85,B 0,C 180,E1 -424.274,E2 -424.274} C_VEL
LIN {X 0,Y 608.461,Z 531.392,A -85,B 0,C 180,E1 -426.877,E2 -426.877} C_VEL
LIN {X 0,Y 608.46,Z 539.883,A -85,B 0,C 180,E1 -429.323,E2 -429.323} C_VEL
LIN {X 0,Y 608.442,Z 549.959,A -85,B 0,C 180,E1 -432.176,E2 -432.176} C_VEL
LIN {X 0,Y 608.459,Z 554.427,A -85,B 0,C 180,E1 -433.427,E2 -433.427} C_VEL
LIN {X 0,Y 608.687,Z 568.619,A -85,B 0,C 180,E1 -433.646,E2 -433.646} C_VEL
LIN {X 0,Y 608.634,Z 583.766,A -85,B 0,C 180,E1 -433.997,E2 -433.997} C_VEL
LIN {X 0,Y 608.625,Z 598.304,A -85,B 0,C 180,E1 -434.469,E2 -434.469} C_VEL
LIN {X 0,Y 608.591,Z 611.613,A -85,B 0,C 180,E1 -435.026,E2 -435.026} C_VEL
LIN {X 0,Y 608.569,Z 624.788,A -85,B 0,C 180,E1 -435.709,E2 -435.709} C_VEL
LIN {X 0,Y 608.548,Z 638.199,A -85,B 0,C 180,E1 -436.56,E2 -436.56} C_VEL
LIN {X 0,Y 608.504,Z 650.387,A -85,B 0,C 180,E1 -437.493,E2 -437.493} C_VEL
LIN {X 0,Y 608.497,Z 661.508,A -85,B 0,C 180,E1 -438.508,E2 -438.508} C_VEL
LIN {X 0,Y 608.476,Z 672.297,A -85,B 0,C 180,E1 -439.687,E2 -439.687} C_VEL
LIN {X 0,Y 608.47,Z 681.289,A -85,B 0,C 180,E1 -440.862,E2 -440.862} C_VEL
LIN {X 0,Y 608.458,Z 688.751,A -85,B 0,C 180,E1 -442.033,E2 -442.033} C_VEL
LIN {X 0,Y 608.44,Z 695.86,A -85,B 0,C 180,E1 -443.399,E2 -443.399} C_VEL
LIN {X 0,Y 608.437,Z 701.16,A -85,B 0,C 180,E1 -444.698,E2 -444.698} C_VEL
LIN {X 0,Y 608.431,Z 705.287,A -85,B 0,C 180,E1 -446.026,E2 -446.026} C_VEL
LIN {X 0,Y 608.423,Z 708.184,A -85,B 0,C 180,E1 -447.351,E2 -447.351} C_VEL
LIN {X 0,Y 608.445,Z 709.912,A -85,B 0,C 180,E1 -448.676,E2 -448.676} C_VEL
LIN {X 0,Y 608.431,Z 710.5,A -85,B 0,C 180,E1 -450,E2 -450} C_VEL
LIN {X 0,Y 608.445,Z 709.912,A -85,B 0,C 180,E1 -451.323,E2 -451.323} C_VEL
LIN {X 0,Y 608.423,Z 708.185,A -85,B 0,C 180,E1 -452.648,E2 -452.648} C_VEL
LIN {X 0,Y 608.431,Z 705.289,A -85,B 0,C 180,E1 -453.974,E2 -453.974} C_VEL
LIN {X 0,Y 608.437,Z 701.163,A -85,B 0,C 180,E1 -455.302,E2 -455.302} C_VEL
LIN {X 0,Y 608.436,Z 695.705,A -85,B 0,C 180,E1 -456.633,E2 -456.633} C_VEL
LIN {X 0,Y 608.457,Z 688.755,A -85,B 0,C 180,E1 -457.967,E2 -457.967} C_VEL
LIN {X 0,Y 608.47,Z 681.293,A -85,B 0,C 180,E1 -459.138,E2 -459.138} C_VEL
LIN {X 0,Y 608.476,Z 672.303,A -85,B 0,C 180,E1 -460.313,E2 -460.313} C_VEL
LIN {X 0,Y 608.496,Z 661.515,A -85,B 0,C 180,E1 -461.492,E2 -461.492} C_VEL
LIN {X 0,Y 608.504,Z 650.396,A -85,B 0,C 180,E1 -462.506,E2 -462.506} C_VEL
LIN {X 0,Y 608.548,Z 638.209,A -85,B 0,C 180,E1 -463.439,E2 -463.439} C_VEL
LIN {X 0,Y 608.575,Z 625.232,A -85,B 0,C 180,E1 -464.265,E2 -464.265} C_VEL
LIN {X 0,Y 608.59,Z 611.626,A -85,B 0,C 180,E1 -464.974,E2 -464.974} C_VEL
LIN {X 0,Y 608.604,Z 597.201,A -85,B 0,C 180,E1 -465.573,E2 -465.573} C_VEL
LIN {X 0,Y 608.639,Z 582.274,A -85,B 0,C 180,E1 -466.045,E2 -466.045} C_VEL
LIN {X 0,Y 608.679,Z 566.948,A -85,B 0,C 180,E1 -466.385,E2 -466.385} C_VEL
LIN {X 0,Y 608.569,Z 555.099,A -85,B 0,C 180,E1 -466.561,E2 -466.561} C_VEL
LIN {X 0,Y 608.453,Z 554.384,A -85,B 0,C 180,E1 -466.585,E2 -466.585} C_VEL
LIN {X 0,Y 608.455,Z 545.01,A -85,B 0,C 180,E1 -469.219,E2 -469.219} C_VEL
LIN {X 0,Y 608.489,Z 535.108,A -85,B 0,C 180,E1 -472.047,E2 -472.047} C_VEL
LIN {X 0,Y 608.471,Z 525.206,A -85,B 0,C 180,E1 -474.934,E2 -474.934} C_VEL
LIN {X 0,Y 608.484,Z 516.541,A -85,B 0,C 180,E1 -477.515,E2 -477.515} C_VEL
LIN {X 0,Y 608.494,Z 508.469,A -85,B 0,C 180,E1 -479.976,E2 -479.976} C_VEL
LIN {X 0,Y 608.519,Z 500.294,A -85,B 0,C 180,E1 -482.531,E2 -482.531} C_VEL
LIN {X 0,Y 608.551,Z 491.785,A -85,B 0,C 180,E1 -485.269,E2 -485.269} C_VEL
LIN {X 0,Y 608.518,Z 484.205,A -85,B 0,C 180,E1 -487.741,E2 -487.741} C_VEL
LIN {X 0,Y 608.533,Z 476.626,A -85,B 0,C 180,E1 -490.338,E2 -490.338} C_VEL
LIN {X 0,Y 608.465,Z 473.319,A -85,B 0,C 180,E1 -491.575,E2 -491.575} C_VEL
LIN {X 0,Y 608.459,Z 473.322,A -85,B 0,C 180,E1 -494.264,E2 -494.264} C_VEL
LIN {X 0,Y 608.455,Z 473.32,A -85,B 0,C 180,E1 -497.041,E2 -497.041} C_VEL
LIN {X 0,Y 608.458,Z 473.321,A -85,B 0,C 180,E1 -499.697,E2 -499.697} C_VEL
LIN {X 0,Y 608.467,Z 473.319,A -85,B 0,C 180,E1 -502.254,E2 -502.254} C_VEL
LIN {X 0,Y 608.48,Z 473.318,A -85,B 0,C 180,E1 -505.088,E2 -505.088} C_VEL
LIN {X 0,Y 608.468,Z 473.318,A -85,B 0,C 180,E1 -507.906,E2 -507.906} C_VEL
LIN {X 0,Y 608.472,Z 473.318,A -85,B 0,C 180,E1 -510.221,E2 -510.221} C_VEL
LIN {X 0,Y 608.479,Z 473.318,A -85,B 0,C 180,E1 -512.79,E2 -512.79} C_VEL
LIN {X 0,Y 608.447,Z 473.322,A -85,B 0,C 180,E1 -515.429,E2 -515.429} C_VEL
LIN {X 0,Y 608.472,Z 473.319,A -85,B 0,C 180,E1 -518.309,E2 -518.309} C_VEL
LIN {X 0,Y 608.471,Z 473.318,A -85,B 0,C 180,E1 -521.28,E2 -521.28} C_VEL
LIN {X 0,Y 608.464,Z 473.32,A -85,B 0,C 180,E1 -523.906,E2 -523.906} C_VEL
LIN {X 0,Y 608.46,Z 473.319,A -85,B 0,C 180,E1 -526.644,E2 -526.644} C_VEL
LIN {X 0,Y 608.467,Z 473.319,A -85,B 0,C 180,E1 -529.35,E2 -529.35} C_VEL
LIN {X 0,Y 608.475,Z 473.318,A -85,B 0,C 180,E1 -532.033,E2 -532.033} C_VEL
LIN {X 0,Y 608.466,Z 473.319,A -85,B 0,C 180,E1 -534.698,E2 -534.698} C_VEL
LIN {X 0,Y 608.485,Z 473.319,A -85,B 0,C 180,E1 -537.352,E2 -537.352} C_VEL
LIN {X 0,Y 608.467,Z 473.318,A -85,B 0,C 180,E1 -540,E2 -540} C_VEL
LIN {X 0,Y 608.483,Z 473.318,A -85,B 0,C 180,E1 -542.648,E2 -542.648} C_VEL
LIN {X 0,Y 608.469,Z 473.319,A -85,B 0,C 180,E1 -545.302,E2 -545.302} C_VEL
LIN {X 0,Y 608.476,Z 473.318,A -85,B 0,C 180,E1 -547.967,E2 -547.967} C_VEL
LIN {X 0,Y 608.453,Z 473.321,A -85,B 0,C 180,E1 -549.473,E2 -549.473} C_VEL
LIN {X 0,Y 607.774,Z 473.405,A -85,B 0,C 180,E1 -550.026,E2 -550.026} C_VEL
LIN {X 0,Y 604.919,Z 473.76,A -85,B 0,C 180,E1 -550.923,E2 -550.923} C_VEL
LIN {X 0,Y 602.516,Z 474.062,A -85,B 0,C 180,E1 -551.644,E2 -551.644} C_VEL
LIN {X 0,Y 601.489,Z 474.187,A -85,B 0,C 180,E1 -552.201,E2 -552.201} C_VEL
LIN {X 0,Y 601.406,Z 474.197,A -85,B 0,C 180,E1 -552.389,E2 -552.389} C_VEL
LIN {X 0,Y 601.43,Z 474.198,A -85,B 0,C 180,E1 -554.897,E2 -554.897} C_VEL
LIN {X 0,Y 601.431,Z 474.197,A -85,B 0,C 180,E1 -556.986,E2 -556.986} C_VEL
LIN {X 0,Y 601.407,Z 474.198,A -85,B 0,C 180,E1 -559.81,E2 -559.81} C_VEL
LIN {X 0,Y 601.404,Z 474.2,A -85,B 0,C 180,E1 -562.684,E2 -562.684} C_VEL
LIN {X 0,Y 601.401,Z 474.201,A -85,B 0,C 180,E1 -564.879,E2 -564.879} C_VEL
LIN {X 0,Y 601.422,Z 474.197,A -85,B 0,C 180,E1 -567.868,E2 -567.868} C_VEL
LIN {X 0,Y 601.442,Z 474.195,A -85,B 0,C 180,E1 -570.164,E2 -570.164} C_VEL
LIN {X 0,Y 601.422,Z 474.197,A -85,B 0,C 180,E1 -572.718,E2 -572.718} C_VEL
LIN {X 0,Y 601.415,Z 474.197,A -85,B 0,C 180,E1 -575.117,E2 -575.117} C_VEL
LIN {X 0,Y 601.432,Z 474.195,A -85,B 0,C 180,E1 -577.42,E2 -577.42} C_VEL
LIN {X 0,Y 601.413,Z 474.198,A -85,B 0,C 180,E1 -579.995,E2 -579.995} C_VEL
LIN {X 0,Y 601.412,Z 474.198,A -85,B 0,C 180,E1 -582.671,E2 -582.671} C_VEL
LIN {X 0,Y 601.422,Z 474.197,A -85,B 0,C 180,E1 -585.483,E2 -585.483} C_VEL
LIN {X 0,Y 601.427,Z 474.195,A -85,B 0,C 180,E1 -588.407,E2 -588.407} C_VEL
LIN {X 0,Y 601.437,Z 474.194,A -85,B 0,C 180,E1 -590.877,E2 -590.877} C_VEL
LIN {X 0,Y 601.444,Z 474.194,A -85,B 0,C 180,E1 -593.735,E2 -593.735} C_VEL
LIN {X 0,Y 601.426,Z 474.198,A -85,B 0,C 180,E1 -596.688,E2 -596.688} C_VEL
LIN {X 0,Y 601.434,Z 474.196,A -85,B 0,C 180,E1 -599.06,E2 -599.06} C_VEL
LIN {X 0,Y 601.436,Z 474.195,A -85,B 0,C 180,E1 -601.374,E2 -601.374} C_VEL
LIN {X 0,Y 601.409,Z 474.198,A -85,B 0,C 180,E1 -603.637,E2 -603.637} C_VEL
LIN {X 0,Y 601.423,Z 474.198,A -85,B 0,C 180,E1 -606.591,E2 -606.591} C_VEL
LIN {X 0,Y 601.427,Z 474.195,A -85,B 0,C 180,E1 -609.479,E2 -609.479} C_VEL
LIN {X 0,Y 601.401,Z 474.2,A -85,B 0,C 180,E1 -612.312,E2 -612.312} C_VEL
LIN {X 0,Y 601.421,Z 474.199,A -85,B 0,C 180,E1 -614.41,E2 -614.41} C_VEL
LIN {X 0,Y 601.42,Z 474.196,A -85,B 0,C 180,E1 -617.172,E2 -617.172} C_VEL
LIN {X 0,Y 601.432,Z 474.197,A -85,B 0,C 180,E1 -619.905,E2 -619.905} C_VEL
LIN {X 0,Y 601.445,Z 474.193,A -85,B 0,C 180,E1 -622.615,E2 -622.615} C_VEL
LIN {X 0,Y 601.43,Z 474.197,A -85,B 0,C 180,E1 -625.308,E2 -625.308} C_VEL
LIN {X 0,Y 601.436,Z 474.194,A -85,B 0,C 180,E1 -627.991,E2 -627.991} C_VEL
LIN {X 0,Y 601.453,Z 474.193,A -85,B 0,C 180,E1 -630.67,E2 -630.67} C_VEL
LIN {X 0,Y 601.433,Z 474.198,A -85,B 0,C 180,E1 -632.009,E2 -632.009} C_VEL
LIN {X 0,Y 601.38,Z 475.967,A -85,B 0,C 180,E1 -634.021,E2 -634.021} C_VEL
LIN {X 0,Y 601.357,Z 478.7,A -85,B 0,C 180,E1 -636.712,E2 -636.712} C_VEL
LIN {X 0,Y 601.335,Z 481.715,A -85,B 0,C 180,E1 -639.417,E2 -639.417} C_VEL
LIN {X 0,Y 601.349,Z 484.836,A -85,B 0,C 180,E1 -642.144,E2 -642.144} C_VEL
LIN {X 0,Y 601.346,Z 488.073,A -85,B 0,C 180,E1 -644.899,E2 -644.899} C_VEL
LIN {X 0,Y 601.334,Z 490.577,A -85,B 0,C 180,E1 -646.989,E2 -646.989} C_VEL
LIN {X 0,Y 601.315,Z 494.023,A -85,B 0,C 180,E1 -649.813,E2 -649.813} C_VEL
LIN {X 0,Y 601.319,Z 497.595,A -85,B 0,C 180,E1 -652.687,E2 -652.687} C_VEL
LIN {X 0,Y 601.334,Z 498.506,A -85,B 0,C 180,E1 -653.323,E2 -653.323} C_VEL
LIN {X 0,Y 601.871,Z 502.211,A -85,B 0,C 180,E1 -653.392,E2 -653.392} C_VEL
LIN {X 0,Y 601.86,Z 517.347,A -85,B 0,C 180,E1 -653.689,E2 -653.689} C_VEL
LIN {X 0,Y 601.763,Z 532.558,A -85,B 0,C 180,E1 -654.127,E2 -654.127} C_VEL
LIN {X 0,Y 601.743,Z 547.445,A -85,B 0,C 180,E1 -654.708,E2 -654.708} C_VEL
LIN {X 0,Y 601.641,Z 561.837,A -85,B 0,C 180,E1 -655.422,E2 -655.422} C_VEL
LIN {X 0,Y 601.59,Z 574.857,A -85,B 0,C 180,E1 -656.22,E2 -656.22} C_VEL
LIN {X 0,Y 601.524,Z 586.905,A -85,B 0,C 180,E1 -657.107,E2 -657.107} C_VEL
LIN {X 0,Y 601.481,Z 597.75,A -85,B 0,C 180,E1 -658.054,E2 -658.054} C_VEL
LIN {X 0,Y 601.456,Z 607.534,A -85,B 0,C 180,E1 -659.057,E2 -659.057} C_VEL
LIN {X 0,Y 601.412,Z 616.707,A -85,B 0,C 180,E1 -660.165,E2 -660.165} C_VEL
LIN {X 0,Y 601.383,Z 625.55,A -85,B 0,C 180,E1 -661.448,E2 -661.448} C_VEL
LIN {X 0,Y 601.367,Z 632.679,A -85,B 0,C 180,E1 -662.706,E2 -662.706} C_VEL
LIN {X 0,Y 601.344,Z 639.097,A -85,B 0,C 180,E1 -664.123,E2 -664.123} C_VEL
LIN {X 0,Y 601.323,Z 642.592,A -85,B 0,C 180,E1 -665.101,E2 -665.101} C_VEL
LIN {X 0,Y 601.316,Z 645.882,A -85,B 0,C 180,E1 -666.249,E2 -666.249} C_VEL
LIN {X 0,Y 601.329,Z 648.285,A -85,B 0,C 180,E1 -667.426,E2 -667.426} C_VEL
LIN {X 0,Y 601.313,Z 649.681,A -85,B 0,C 180,E1 -668.456,E2 -668.456} C_VEL
LIN {X 0,Y 601.301,Z 650.496,A -85,B 0,C 180,E1 -670.003,E2 -670.003} C_VEL
LIN {X 0,Y 601.322,Z 649.743,A -85,B 0,C 180,E1 -671.581,E2 -671.581} C_VEL
LIN {X 0,Y 601.341,Z 648.265,A -85,B 0,C 180,E1 -672.676,E2 -672.676} C_VEL
LIN {X 0,Y 601.353,Z 645.313,A -85,B 0,C 180,E1 -674.057,E2 -674.057} C_VEL
LIN {X 0,Y 601.335,Z 640.929,A -85,B 0,C 180,E1 -675.473,E2 -675.473} C_VEL
LIN {X 0,Y 601.367,Z 635.102,A -85,B 0,C 180,E1 -676.882,E2 -676.882} C_VEL
LIN {X 0,Y 601.384,Z 628.009,A -85,B 0,C 180,E1 -678.231,E2 -678.231} C_VEL
LIN {X 0,Y 601.403,Z 620.338,A -85,B 0,C 180,E1 -679.427,E2 -679.427} C_VEL
LIN {X 0,Y 601.45,Z 610.707,A -85,B 0,C 180,E1 -680.67,E2 -680.67} C_VEL
LIN {X 0,Y 601.5,Z 599.744,A -85,B 0,C 180,E1 -681.844,E2 -681.844} C_VEL
LIN {X 0,Y 601.531,Z 587.824,A -85,B 0,C 180,E1 -682.908,E2 -682.908} C_VEL
LIN {X 0,Y 601.622,Z 576.061,A -85,B 0,C 180,E1 -683.788,E2 -683.788} C_VEL
LIN {X 0,Y 601.658,Z 563.069,A -85,B 0,C 180,E1 -684.599,E2 -684.599} C_VEL
LIN {X 0,Y 601.707,Z 549.544,A -85,B 0,C 180,E1 -685.291,E2 -685.291} C_VEL
LIN {X 0,Y 601.775,Z 535.798,A -85,B 0,C 180,E1 -685.853,E2 -685.853} C_VEL
LIN {X 0,Y 601.843,Z 520.105,A -85,B 0,C 180,E1 -686.336,E2 -686.336} C_VEL
LIN {X 0,Y 601.898,Z 505.224,A -85,B 0,C 180,E1 -686.653,E2 -686.653} C_VEL
LIN {X 0,Y 601.734,Z 500.561,A -85,B 0,C 180,E1 -686.726,E2 -686.726} C_VEL
LIN {X 0,Y 601.335,Z 498.37,A -85,B 0,C 180,E1 -686.785,E2 -686.785} C_VEL
LIN {X 0,Y 601.344,Z 494.532,A -85,B 0,C 180,E1 -689.864,E2 -689.864} C_VEL
LIN {X 0,Y 601.339,Z 491.122,A -85,B 0,C 180,E1 -692.65,E2 -692.65} C_VEL
LIN {X 0,Y 601.344,Z 488.159,A -85,B 0,C 180,E1 -695.118,E2 -695.118} C_VEL
LIN {X 0,Y 601.334,Z 484.731,A -85,B 0,C 180,E1 -698.037,E2 -698.037} C_VEL
LIN {X 0,Y 601.332,Z 482.264,A -85,B 0,C 180,E1 -700.188,E2 -700.188} C_VEL
LIN {X 0,Y 601.362,Z 479.879,A -85,B 0,C 180,E1 -702.31,E2 -702.31} C_VEL
LIN {X 0,Y 601.373,Z 477.803,A -85,B 0,C 180,E1 -704.407,E2 -704.407} C_VEL
LIN {X 0,Y 601.372,Z 475.666,A -85,B 0,C 180,E1 -706.483,E2 -706.483} C_VEL
LIN {X 0,Y 601.385,Z 474.315,A -85,B 0,C 180,E1 -707.857,E2 -707.857} C_VEL
LIN {X 0,Y 601.44,Z 474.193,A -85,B 0,C 180,E1 -709.905,E2 -709.905} C_VEL
LIN {X 0,Y 601.438,Z 474.189,A -85,B 0,C 180,E1 -712.615,E2 -712.615} C_VEL
LIN {X 0,Y 601.429,Z 474.19,A -85,B 0,C 180,E1 -715.308,E2 -715.308} C_VEL
LIN {X 0,Y 601.426,Z 474.194,A -85,B 0,C 180,E1 -717.991,E2 -717.991} C_VEL
LIN {X 0,Y 601.45,Z 474.186,A -85,B 0,C 180,E1 -720.669,E2 -720.669} C_VEL
LIN {X 0,Y 601.427,Z 474.197,A -85,B 0,C 180,E1 -723.349,E2 -723.349} C_VEL
LIN {X 0,Y 601.407,Z 474.191,A -85,B 0,C 180,E1 -726.037,E2 -726.037} C_VEL
LIN {X 0,Y 601.438,Z 474.191,A -85,B 0,C 180,E1 -728.737,E2 -728.737} C_VEL
LIN {X 0,Y 601.429,Z 474.191,A -85,B 0,C 180,E1 -731.458,E2 -731.458} C_VEL
LIN {X 0,Y 601.415,Z 474.191,A -85,B 0,C 180,E1 -734.205,E2 -734.205} C_VEL
LIN {X 0,Y 601.43,Z 474.193,A -85,B 0,C 180,E1 -736.986,E2 -736.986} C_VEL
LIN {X 0,Y 601.402,Z 474.192,A -85,B 0,C 180,E1 -739.809,E2 -739.809} C_VEL
LIN {X 0,Y 601.412,Z 474.197,A -85,B 0,C 180,E1 -742.606,E2 -742.606} C_VEL
LIN {X 0,Y 601.401,Z 474.193,A -85,B 0,C 180,E1 -744.878,E2 -744.878} C_VEL
LIN {X 0,Y 601.422,Z 474.195,A -85,B 0,C 180,E1 -747.867,E2 -747.867} C_VEL
LIN {X 0,Y 601.445,Z 474.194,A -85,B 0,C 180,E1 -750.163,E2 -750.163} C_VEL
LIN {X 0,Y 601.421,Z 474.19,A -85,B 0,C 180,E1 -752.716,E2 -752.716} C_VEL
LIN {X 0,Y 601.415,Z 474.191,A -85,B 0,C 180,E1 -755.115,E2 -755.115} C_VEL
LIN {X 0,Y 601.431,Z 474.195,A -85,B 0,C 180,E1 -757.419,E2 -757.419} C_VEL
LIN {X 0,Y 601.409,Z 474.193,A -85,B 0,C 180,E1 -759.995,E2 -759.995} C_VEL
LIN {X 0,Y 601.41,Z 474.192,A -85,B 0,C 180,E1 -762.67,E2 -762.67} C_VEL
LIN {X 0,Y 601.423,Z 474.195,A -85,B 0,C 180,E1 -765.482,E2 -765.482} C_VEL
LIN {X 0,Y 601.439,Z 474.295,A -85,B 0,C 180,E1 -768.293,E2 -768.293} C_VEL
LIN {X 0,Y 601.61,Z 479.016,A -85,B 0,C 180,E1 -770.021,E2 -770.021} C_VEL
LIN {X 0,Y 601.561,Z 486.499,A -85,B 0,C 180,E1 -772.602,E2 -772.602} C_VEL
LIN {X 0,Y 601.522,Z 494.14,A -85,B 0,C 180,E1 -775.076,E2 -775.076} C_VEL
LIN {X 0,Y 601.53,Z 501.685,A -85,B 0,C 180,E1 -777.491,E2 -777.491} C_VEL
LIN {X 0,Y 601.489,Z 510.35,A -85,B 0,C 180,E1 -780.226,E2 -780.226} C_VEL
LIN {X 0,Y 601.457,Z 519.014,A -85,B 0,C 180,E1 -782.889,E2 -782.889} C_VEL
LIN {X 0,Y 601.454,Z 526.441,A -85,B 0,C 180,E1 -785.124,E2 -785.124} C_VEL
LIN {X 0,Y 601.439,Z 536.343,A -85,B 0,C 180,E1 -788.042,E2 -788.042} C_VEL
LIN {X 0,Y 601.407,Z 546.245,A -85,B 0,C 180,E1 -790.901,E2 -790.901} C_VEL
LIN {X 0,Y 601.387,Z 554.387,A -85,B 0,C 180,E1 -793.215,E2 -793.215} C_VEL
LIN {X 0,Y 601.888,Z 558.673,A -85,B 0,C 180,E1 -793.296,E2 -793.296} C_VEL
LIN {X 0,Y 601.849,Z 573.761,A -85,B 0,C 180,E1 -793.558,E2 -793.558} C_VEL
LIN {X 0,Y 601.798,Z 588.297,A -85,B 0,C 180,E1 -793.941,E2 -793.941} C_VEL
LIN {X 0,Y 601.769,Z 602.79,A -85,B 0,C 180,E1 -794.462,E2 -794.462} C_VEL
LIN {X 0,Y 601.683,Z 616.86,A -85,B 0,C 180,E1 -795.109,E2 -795.109} C_VEL
LIN {X 0,Y 601.614,Z 630.582,A -85,B 0,C 180,E1 -795.894,E2 -795.894} C_VEL
LIN {X 0,Y 601.57,Z 644.012,A -85,B 0,C 180,E1 -796.832,E2 -796.832} C_VEL
LIN {X 0,Y 601.514,Z 656.191,A -85,B 0,C 180,E1 -797.859,E2 -797.859} C_VEL
LIN {X 0,Y 601.437,Z 667.272,A -85,B 0,C 180,E1 -798.982,E2 -798.982} C_VEL
LIN {X 0,Y 601.427,Z 676.369,A -85,B 0,C 180,E1 -800.075,E2 -800.075} C_VEL
LIN {X 0,Y 601.387,Z 684.653,A -85,B 0,C 180,E1 -801.261,E2 -801.261} C_VEL
LIN {X 0,Y 601.366,Z 692.425,A -85,B 0,C 180,E1 -802.614,E2 -802.614} C_VEL
LIN {X 0,Y 601.352,Z 698.606,A -85,B 0,C 180,E1 -803.962,E2 -803.962} C_VEL
LIN {X 0,Y 601.33,Z 703.382,A -85,B 0,C 180,E1 -805.307,E2 -805.307} C_VEL
LIN {X 0,Y 601.337,Z 706.885,A -85,B 0,C 180,E1 -806.65,E2 -806.65} C_VEL
LIN {X 0,Y 601.339,Z 709.191,A -85,B 0,C 180,E1 -807.99,E2 -807.99} C_VEL
LIN {X 0,Y 601.337,Z 710.35,A -85,B 0,C 180,E1 -809.33,E2 -809.33} C_VEL
LIN {X 0,Y 601.336,Z 710.35,A -85,B 0,C 180,E1 -810.669,E2 -810.669} C_VEL
LIN {X 0,Y 601.339,Z 709.192,A -85,B 0,C 180,E1 -812.009,E2 -812.009} C_VEL
LIN {X 0,Y 601.337,Z 706.887,A -85,B 0,C 180,E1 -813.35,E2 -813.35} C_VEL
LIN {X 0,Y 601.33,Z 703.384,A -85,B 0,C 180,E1 -814.692,E2 -814.692} C_VEL
LIN {X 0,Y 601.352,Z 698.61,A -85,B 0,C 180,E1 -816.037,E2 -816.037} C_VEL
LIN {X 0,Y 601.382,Z 692.428,A -85,B 0,C 180,E1 -817.385,E2 -817.385} C_VEL
LIN {X 0,Y 601.387,Z 684.657,A -85,B 0,C 180,E1 -818.738,E2 -818.738} C_VEL
LIN {X 0,Y 601.427,Z 676.374,A -85,B 0,C 180,E1 -819.925,E2 -819.925} C_VEL
LIN {X 0,Y 601.46,Z 665.935,A -85,B 0,C 180,E1 -821.164,E2 -821.164} C_VEL
LIN {X 0,Y 601.513,Z 656.198,A -85,B 0,C 180,E1 -822.14,E2 -822.14} C_VEL
LIN {X 0,Y 601.57,Z 644.023,A -85,B 0,C 180,E1 -823.168,E2 -823.168} C_VEL
LIN {X 0,Y 601.605,Z 632.087,A -85,B 0,C 180,E1 -824.011,E2 -824.011} C_VEL
LIN {X 0,Y 601.665,Z 618.539,A -85,B 0,C 180,E1 -824.804,E2 -824.804} C_VEL
LIN {X 0,Y 601.761,Z 603.858,A -85,B 0,C 180,E1 -825.495,E2 -825.495} C_VEL
LIN {X 0,Y 601.782,Z 589.637,A -85,B 0,C 180,E1 -826.015,E2 -826.015} C_VEL
LIN {X 0,Y 601.855,Z 574.655,A -85,B 0,C 180,E1 -826.421,E2 -826.421} C_VEL
LIN {X 0,Y 601.886,Z 559.274,A -85,B 0,C 180,E1 -826.695,E2 -826.695} C_VEL
LIN {X 0,Y 601.456,Z 554.945,A -85,B 0,C 180,E1 -826.765,E2 -826.765} C_VEL
LIN {X 0,Y 601.391,Z 554.285,A -85,B 0,C 180,E1 -826.814,E2 -826.814} C_VEL
LIN {X 0,Y 601.418,Z 545.01,A -85,B 0,C 180,E1 -829.453,E2 -829.453} C_VEL
LIN {X 0,Y 601.455,Z 535.239,A -85,B 0,C 180,E1 -832.28,E2 -832.28} C_VEL
LIN {X 0,Y 601.453,Z 525.206,A -85,B 0,C 180,E1 -835.245,E2 -835.245} C_VEL
LIN {X 0,Y 601.508,Z 516.541,A -85,B 0,C 180,E1 -837.862,E2 -837.862} C_VEL
LIN {X 0,Y 601.5,Z 507.877,A -85,B 0,C 180,E1 -840.547,E2 -840.547} C_VEL
LIN {X 0,Y 601.557,Z 499.212,A -85,B 0,C 180,E1 -843.304,E2 -843.304} C_VEL
LIN {X 0,Y 601.563,Z 491.631,A -85,B 0,C 180,E1 -845.741,E2 -845.741} C_VEL
LIN {X 0,Y 601.594,Z 483.427,A -85,B 0,C 180,E1 -848.491,E2 -848.491} C_VEL
LIN {X 0,Y 601.632,Z 475.697,A -85,B 0,C 180,E1 -851.222,E2 -851.222} C_VEL
LIN {X 0,Y 601.436,Z 474.195,A -85,B 0,C 180,E1 -851.819,E2 -851.819} C_VEL
LIN {X 0,Y 601.417,Z 474.198,A -85,B 0,C 180,E1 -854.535,E2 -854.535} C_VEL
LIN {X 0,Y 601.435,Z 474.195,A -85,B 0,C 180,E1 -857.405,E2 -857.405} C_VEL
LIN {X 0,Y 601.443,Z 474.193,A -85,B 0,C 180,E1 -860.462,E2 -860.462} C_VEL
LIN {X 0,Y 601.409,Z 474.198,A -85,B 0,C 180,E1 -863.418,E2 -863.418} C_VEL
LIN {X 0,Y 601.432,Z 474.195,A -85,B 0,C 180,E1 -866.062,E2 -866.062} C_VEL
LIN {X 0,Y 601.436,Z 474.196,A -85,B 0,C 180,E1 -868.541,E2 -868.541} C_VEL
LIN {X 0,Y 601.434,Z 474.194,A -85,B 0,C 180,E1 -871.373,E2 -871.373} C_VEL
LIN {X 0,Y 601.415,Z 474.2,A -85,B 0,C 180,E1 -874.129,E2 -874.129} C_VEL
LIN {X 0,Y 601.416,Z 474.198,A -85,B 0,C 180,E1 -876.59,E2 -876.59} C_VEL
LIN {X 0,Y 601.432,Z 474.196,A -85,B 0,C 180,E1 -879.478,E2 -879.478} C_VEL
LIN {X 0,Y 601.394,Z 474.199,A -85,B 0,C 180,E1 -882.312,E2 -882.312} C_VEL
LIN {X 0,Y 601.412,Z 474.197,A -85,B 0,C 180,E1 -884.409,E2 -884.409} C_VEL
LIN {X 0,Y 601.42,Z 474.197,A -85,B 0,C 180,E1 -887.172,E2 -887.172} C_VEL
LIN {X 0,Y 601.431,Z 474.195,A -85,B 0,C 180,E1 -889.905,E2 -889.905} C_VEL
LIN {X 0,Y 601.45,Z 474.193,A -85,B 0,C 180,E1 -892.615,E2 -892.615} C_VEL
LIN {X 0,Y 601.428,Z 474.196,A -85,B 0,C 180,E1 -895.308,E2 -895.308} C_VEL
LIN {X 0,Y 601.421,Z 474.196,A -85,B 0,C 180,E1 -897.991,E2 -897.991} C_VEL
LIN {X 0,Y 601.451,Z 474.194,A -85,B 0,C 180,E1 -900.67,E2 -900.67} C_VEL
LIN {X 0,Y 601.432,Z 474.195,A -85,B 0,C 180,E1 -903.35,E2 -903.35} C_VEL
LIN {X 0,Y 601.437,Z 474.197,A -85,B 0,C 180,E1 -906.037,E2 -906.037} C_VEL
LIN {X 0,Y 601.437,Z 474.194,A -85,B 0,C 180,E1 -908.738,E2 -908.738} C_VEL
LIN {X 0,Y 601.426,Z 474.197,A -85,B 0,C 180,E1 -911.459,E2 -911.459} C_VEL
LIN {X 0,Y 601.406,Z 474.197,A -85,B 0,C 180,E1 -912.389,E2 -912.389} C_VEL
LIN {X 0,Y 600.745,Z 474.282,A -85,B 0,C 180,E1 -912.949,E2 -912.949} C_VEL
LIN {X 0,Y 597.894,Z 474.638,A -85,B 0,C 180,E1 -913.857,E2 -913.857} C_VEL
LIN {X 0,Y 595.483,Z 474.937,A -85,B 0,C 180,E1 -914.587,E2 -914.587} C_VEL
LIN {X 0,Y 594.447,Z 475.066,A -85,B 0,C 180,E1 -915.15,E2 -915.15} C_VEL
LIN {X 0,Y 594.362,Z 475.075,A -85,B 0,C 180,E1 -915.341,E2 -915.341} C_VEL
LIN {X 0,Y 594.38,Z 475.074,A -85,B 0,C 180,E1 -917.905,E2 -917.905} C_VEL
LIN {X 0,Y 594.378,Z 475.073,A -85,B 0,C 180,E1 -920.92,E2 -920.92} C_VEL
LIN {X 0,Y 594.386,Z 475.075,A -85,B 0,C 180,E1 -923.705,E2 -923.705} C_VEL
LIN {X 0,Y 594.387,Z 475.072,A -85,B 0,C 180,E1 -926.7,E2 -926.7} C_VEL
LIN {X 0,Y 594.38,Z 475.074,A -85,B 0,C 180,E1 -928.999,E2 -928.999} C_VEL
LIN {X 0,Y 594.389,Z 475.073,A -85,B 0,C 180,E1 -931.647,E2 -931.647} C_VEL
LIN {X 0,Y 594.394,Z 475.073,A -85,B 0,C 180,E1 -934.579,E2 -934.579} C_VEL
LIN {X 0,Y 594.384,Z 475.074,A -85,B 0,C 180,E1 -937.087,E2 -937.087} C_VEL
LIN {X 0,Y 594.378,Z 475.073,A -85,B 0,C 180,E1 -939.776,E2 -939.776} C_VEL
LIN {X 0,Y 594.37,Z 475.077,A -85,B 0,C 180,E1 -942.376,E2 -942.376} C_VEL
LIN {X 0,Y 594.36,Z 475.075,A -85,B 0,C 180,E1 -945.192,E2 -945.192} C_VEL
LIN {X 0,Y 594.37,Z 475.075,A -85,B 0,C 180,E1 -947.626,E2 -947.626} C_VEL
LIN {X 0,Y 594.393,Z 475.073,A -85,B 0,C 180,E1 -950.322,E2 -950.322} C_VEL
LIN {X 0,Y 594.387,Z 475.072,A -85,B 0,C 180,E1 -952.915,E2 -952.915} C_VEL
LIN {X 0,Y 594.381,Z 475.074,A -85,B 0,C 180,E1 -955.862,E2 -955.862} C_VEL
LIN {X 0,Y 594.391,Z 475.072,A -85,B 0,C 180,E1 -958.652,E2 -958.652} C_VEL
LIN {X 0,Y 594.385,Z 475.074,A -85,B 0,C 180,E1 -961.043,E2 -961.043} C_VEL
LIN {X 0,Y 594.393,Z 475.071,A -85,B 0,C 180,E1 -963.977,E2 -963.977} C_VEL
LIN {X 0,Y 594.395,Z 475.072,A -85,B 0,C 180,E1 -966.297,E2 -966.297} C_VEL
LIN {X 0,Y 594.4,Z 475.071,A -85,B 0,C 180,E1 -969.225,E2 -969.225} C_VEL
LIN {X 0,Y 594.383,Z 475.075,A -85,B 0,C 180,E1 -972.097,E2 -972.097} C_VEL
LIN {X 0,Y 594.374,Z 475.076,A -85,B 0,C 180,E1 -974.22,E2 -974.22} C_VEL
LIN {X 0,Y 594.387,Z 475.073,A -85,B 0,C 180,E1 -976.322,E2 -976.322} C_VEL
LIN {X 0,Y 594.378,Z 475.074,A -85,B 0,C 180,E1 -979.095,E2 -979.095} C_VEL
LIN {X 0,Y 594.387,Z 475.073,A -85,B 0,C 180,E1 -981.843,E2 -981.843} C_VEL
LIN {X 0,Y 594.395,Z 475.072,A -85,B 0,C 180,E1 -984.573,E2 -984.573} C_VEL
LIN {X 0,Y 594.408,Z 475.07,A -85,B 0,C 180,E1 -987.29,E2 -987.29} C_VEL
LIN {X 0,Y 594.42,Z 475.069,A -85,B 0,C 180,E1 -990,E2 -990} C_VEL
LIN {X 0,Y 594.4,Z 475.074,A -85,B 0,C 180,E1 -992.033,E2 -992.033} C_VEL
LIN {X 0,Y 594.293,Z 475.247,A -85,B 0,C 180,E1 -992.712,E2 -992.712} C_VEL
LIN {X 0,Y 594.297,Z 477.993,A -85,B 0,C 180,E1 -995.429,E2 -995.429} C_VEL
LIN {X 0,Y 594.279,Z 480.768,A -85,B 0,C 180,E1 -998.159,E2 -998.159} C_VEL
LIN {X 0,Y 594.286,Z 483.967,A -85,B 0,C 180,E1 -1001.02,E2 -1001.02} C_VEL
LIN {X 0,Y 594.283,Z 487.548,A -85,B 0,C 180,E1 -1004.131,E2 -1004.131} C_VEL
LIN {X 0,Y 594.242,Z 490.543,A -85,B 0,C 180,E1 -1006.668,E2 -1006.668} C_VEL
LIN {X 0,Y 594.24,Z 493.754,A -85,B 0,C 180,E1 -1009.339,E2 -1009.339} C_VEL
LIN {X 0,Y 594.254,Z 497.303,A -85,B 0,C 180,E1 -1012.238,E2 -1012.238} C_VEL
LIN {X 0,Y 594.249,Z 498.384,A -85,B 0,C 180,E1 -1013.11,E2 -1013.11} C_VEL
LIN {X 0,Y 595.065,Z 503.5,A -85,B 0,C 180,E1 -1013.214,E2 -1013.214} C_VEL
LIN {X 0,Y 595.045,Z 518.128,A -85,B 0,C 180,E1 -1013.515,E2 -1013.515} C_VEL
LIN {X 0,Y 594.918,Z 533.146,A -85,B 0,C 180,E1 -1013.959,E2 -1013.959} C_VEL
LIN {X 0,Y 594.869,Z 547.629,A -85,B 0,C 180,E1 -1014.534,E2 -1014.534} C_VEL
LIN {X 0,Y 594.735,Z 560.549,A -85,B 0,C 180,E1 -1015.177,E2 -1015.177} C_VEL
LIN {X 0,Y 594.646,Z 573.881,A -85,B 0,C 180,E1 -1015.989,E2 -1015.989} C_VEL
LIN {X 0,Y 594.577,Z 586.007,A -85,B 0,C 180,E1 -1016.88,E2 -1016.88} C_VEL
LIN {X 0,Y 594.484,Z 597.117,A -85,B 0,C 180,E1 -1017.849,E2 -1017.849} C_VEL
LIN {X 0,Y 594.432,Z 608.136,A -85,B 0,C 180,E1 -1018.996,E2 -1018.996} C_VEL
LIN {X 0,Y 594.37,Z 616.73,A -85,B 0,C 180,E1 -1020.049,E2 -1020.049} C_VEL
LIN {X 0,Y 594.312,Z 625.601,A -85,B 0,C 180,E1 -1021.353,E2 -1021.353} C_VEL
LIN {X 0,Y 594.287,Z 632.166,A -85,B 0,C 180,E1 -1022.522,E2 -1022.522} C_VEL
LIN {X 0,Y 594.276,Z 637.908,A -85,B 0,C 180,E1 -1023.768,E2 -1023.768} C_VEL
LIN {X 0,Y 594.239,Z 642.295,A -85,B 0,C 180,E1 -1024.947,E2 -1024.947} C_VEL
LIN {X 0,Y 594.221,Z 646.477,A -85,B 0,C 180,E1 -1026.461,E2 -1026.461} C_VEL
LIN {X 0,Y 594.217,Z 649.125,A -85,B 0,C 180,E1 -1027.953,E2 -1027.953} C_VEL
LIN {X 0,Y 594.206,Z 650.001,A -85,B 0,C 180,E1 -1028.818,E2 -1028.818} C_VEL
LIN {X 0,Y 594.222,Z 650.44,A -85,B 0,C 180,E1 -1029.756,E2 -1029.756} C_VEL
LIN {X 0,Y 594.215,Z 650.321,A -85,B 0,C 180,E1 -1030.803,E2 -1030.803} C_VEL
LIN {X 0,Y 594.253,Z 648.789,A -85,B 0,C 180,E1 -1032.385,E2 -1032.385} C_VEL
LIN {X 0,Y 594.251,Z 646.037,A -85,B 0,C 180,E1 -1033.827,E2 -1033.827} C_VEL
LIN {X 0,Y 594.263,Z 642.115,A -85,B 0,C 180,E1 -1035.201,E2 -1035.201} C_VEL
LIN {X 0,Y 594.3,Z 636.356,A -85,B 0,C 180,E1 -1036.694,E2 -1036.694} C_VEL
LIN {X 0,Y 594.287,Z 630.339,A -85,B 0,C 180,E1 -1037.913,E2 -1037.913} C_VEL
LIN {X 0,Y 594.32,Z 622.722,A -85,B 0,C 180,E1 -1039.184,E2 -1039.184} C_VEL
LIN {X 0,Y 594.397,Z 614.547,A -85,B 0,C 180,E1 -1040.321,E2 -1040.321} C_VEL
LIN {X 0,Y 594.449,Z 604.804,A -85,B 0,C 180,E1 -1041.463,E2 -1041.463} C_VEL
LIN {X 0,Y 594.509,Z 593.884,A -85,B 0,C 180,E1 -1042.539,E2 -1042.539} C_VEL
LIN {X 0,Y 594.601,Z 582.453,A -85,B 0,C 180,E1 -1043.488,E2 -1043.488} C_VEL
LIN {X 0,Y 594.698,Z 569.166,A -85,B 0,C 180,E1 -1044.406,E2 -1044.406} C_VEL
LIN {X 0,Y 594.79,Z 555.32,A -85,B 0,C 180,E1 -1045.19,E2 -1045.19} C_VEL
LIN {X 0,Y 594.896,Z 541.141,A -85,B 0,C 180,E1 -1045.832,E2 -1045.832} C_VEL
LIN {X 0,Y 594.976,Z 526.706,A -85,B 0,C 180,E1 -1046.34,E2 -1046.34} C_VEL
LIN {X 0,Y 595.045,Z 511.689,A -85,B 0,C 180,E1 -1046.725,E2 -1046.725} C_VEL
LIN {X 0,Y 594.91,Z 501.737,A -85,B 0,C 180,E1 -1046.906,E2 -1046.906} C_VEL
LIN {X 0,Y 594.246,Z 498.37,A -85,B 0,C 180,E1 -1046.991,E2 -1046.991} C_VEL
LIN {X 0,Y 594.238,Z 495.04,A -85,B 0,C 180,E1 -1049.695,E2 -1049.695} C_VEL
LIN {X 0,Y 594.258,Z 491.604,A -85,B 0,C 180,E1 -1052.533,E2 -1052.533} C_VEL
LIN {X 0,Y 594.275,Z 487.982,A -85,B 0,C 180,E1 -1055.589,E2 -1055.589} C_VEL
LIN {X 0,Y 594.272,Z 484.625,A -85,B 0,C 180,E1 -1058.493,E2 -1058.493} C_VEL
LIN {X 0,Y 594.28,Z 481.379,A -85,B 0,C 180,E1 -1061.379,E2 -1061.379} C_VEL
LIN {X 0,Y 594.307,Z 479.321,A -85,B 0,C 180,E1 -1063.512,E2 -1063.512} C_VEL
LIN {X 0,Y 594.305,Z 476.508,A -85,B 0,C 180,E1 -1066.319,E2 -1066.319} C_VEL
LIN {X 0,Y 594.322,Z 475.14,A -85,B 0,C 180,E1 -1067.71,E2 -1067.71} C_VEL
LIN {X 0,Y 594.398,Z 475.069,A -85,B 0,C 180,E1 -1069.784,E2 -1069.784} C_VEL
LIN {X 0,Y 594.391,Z 475.067,A -85,B 0,C 180,E1 -1072.526,E2 -1072.526} C_VEL
LIN {X 0,Y 594.398,Z 475.066,A -85,B 0,C 180,E1 -1075.252,E2 -1075.252} C_VEL
LIN {X 0,Y 594.396,Z 475.07,A -85,B 0,C 180,E1 -1077.967,E2 -1077.967} C_VEL
LIN {X 0,Y 594.42,Z 475.062,A -85,B 0,C 180,E1 -1080.677,E2 -1080.677} C_VEL
LIN {X 0,Y 594.379,Z 475.076,A -85,B 0,C 180,E1 -1083.389,E2 -1083.389} C_VEL
LIN {X 0,Y 594.364,Z 475.069,A -85,B 0,C 180,E1 -1086.109,E2 -1086.109} C_VEL
LIN {X 0,Y 594.399,Z 475.069,A -85,B 0,C 180,E1 -1088.842,E2 -1088.842} C_VEL
LIN {X 0,Y 594.389,Z 475.067,A -85,B 0,C 180,E1 -1091.596,E2 -1091.596} C_VEL
LIN {X 0,Y 594.385,Z 475.069,A -85,B 0,C 180,E1 -1094.377,E2 -1094.377} C_VEL
LIN {X 0,Y 594.386,Z 475.068,A -85,B 0,C 180,E1 -1097.193,E2 -1097.193} C_VEL
LIN {X 0,Y 594.373,Z 475.07,A -85,B 0,C 180,E1 -1100.054,E2 -1100.054} C_VEL
LIN {X 0,Y 594.361,Z 475.07,A -85,B 0,C 180,E1 -1102.967,E2 -1102.967} C_VEL
LIN {X 0,Y 594.376,Z 475.067,A -85,B 0,C 180,E1 -1105.193,E2 -1105.193} C_VEL
LIN {X 0,Y 594.381,Z 475.068,A -85,B 0,C 180,E1 -1107.527,E2 -1107.527} C_VEL
LIN {X 0,Y 594.397,Z 475.069,A -85,B 0,C 180,E1 -1110.331,E2 -1110.331} C_VEL
LIN {X 0,Y 594.375,Z 475.067,A -85,B 0,C 180,E1 -1112.95,E2 -1112.95} C_VEL
LIN {X 0,Y 594.382,Z 475.071,A -85,B 0,C 180,E1 -1115.407,E2 -1115.407} C_VEL
LIN {X 0,Y 594.382,Z 475.07,A -85,B 0,C 180,E1 -1117.941,E2 -1117.941} C_VEL
LIN {X 0,Y 594.378,Z 475.068,A -85,B 0,C 180,E1 -1120.823,E2 -1120.823} C_VEL
LIN {X 0,Y 594.38,Z 475.069,A -85,B 0,C 180,E1 -1123.841,E2 -1123.841} C_VEL
LIN {X 0,Y 594.385,Z 475.071,A -85,B 0,C 180,E1 -1126.703,E2 -1126.703} C_VEL
LIN {X 0,Y 594.423,Z 475.242,A -85,B 0,C 180,E1 -1128.065,E2 -1128.065} C_VEL
LIN {X 0,Y 594.658,Z 480.083,A -85,B 0,C 180,E1 -1129.864,E2 -1129.864} C_VEL
LIN {X 0,Y 594.579,Z 487.171,A -85,B 0,C 180,E1 -1132.368,E2 -1132.368} C_VEL
LIN {X 0,Y 594.523,Z 495.216,A -85,B 0,C 180,E1 -1135.039,E2 -1135.039} C_VEL
LIN {X 0,Y 594.567,Z 502.923,A -85,B 0,C 180,E1 -1137.464,E2 -1137.464} C_VEL
LIN {X 0,Y 594.509,Z 511.587,A -85,B 0,C 180,E1 -1140.231,E2 -1140.231} C_VEL
LIN {X 0,Y 594.449,Z 520.252,A -85,B 0,C 180,E1 -1142.924,E2 -1142.924} C_VEL
LIN {X 0,Y 594.436,Z 528.916,A -85,B 0,C 180,E1 -1145.556,E2 -1145.556} C_VEL
LIN {X 0,Y 594.389,Z 538.819,A -85,B 0,C 180,E1 -1148.498,E2 -1148.498} C_VEL
LIN {X 0,Y 594.353,Z 548.721,A -85,B 0,C 180,E1 -1151.382,E2 -1151.382} C_VEL
LIN {X 0,Y 594.328,Z 554.41,A -85,B 0,C 180,E1 -1153.016,E2 -1153.016} C_VEL
LIN {X 0,Y 595.11,Z 558.697,A -85,B 0,C 180,E1 -1153.1,E2 -1153.1} C_VEL
LIN {X 0,Y 595.03,Z 574.025,A -85,B 0,C 180,E1 -1153.37,E2 -1153.37} C_VEL
LIN {X 0,Y 594.974,Z 588.296,A -85,B 0,C 180,E1 -1153.751,E2 -1153.751} C_VEL
LIN {X 0,Y 594.916,Z 602.792,A -85,B 0,C 180,E1 -1154.278,E2 -1154.278} C_VEL
LIN {X 0,Y 594.78,Z 616.862,A -85,B 0,C 180,E1 -1154.933,E2 -1154.933} C_VEL
LIN {X 0,Y 594.683,Z 630.405,A -85,B 0,C 180,E1 -1155.715,E2 -1155.715} C_VEL
LIN {X 0,Y 594.587,Z 642.854,A -85,B 0,C 180,E1 -1156.587,E2 -1156.587} C_VEL
LIN {X 0,Y 594.535,Z 654.274,A -85,B 0,C 180,E1 -1157.541,E2 -1157.541} C_VEL
LIN {X 0,Y 594.434,Z 664.709,A -85,B 0,C 180,E1 -1158.572,E2 -1158.572} C_VEL
LIN {X 0,Y 594.38,Z 675.019,A -85,B 0,C 180,E1 -1159.784,E2 -1159.784} C_VEL
LIN {X 0,Y 594.339,Z 683.532,A -85,B 0,C 180,E1 -1160.986,E2 -1160.986} C_VEL
LIN {X 0,Y 594.311,Z 690.611,A -85,B 0,C 180,E1 -1162.184,E2 -1162.184} C_VEL
LIN {X 0,Y 594.261,Z 697.492,A -85,B 0,C 180,E1 -1163.623,E2 -1163.623} C_VEL
LIN {X 0,Y 594.245,Z 702.323,A -85,B 0,C 180,E1 -1164.911,E2 -1164.911} C_VEL
LIN {X 0,Y 594.253,Z 705.288,A -85,B 0,C 180,E1 -1165.931,E2 -1165.931} C_VEL
LIN {X 0,Y 594.223,Z 708.185,A -85,B 0,C 180,E1 -1167.288,E2 -1167.288} C_VEL
LIN {X 0,Y 594.245,Z 709.912,A -85,B 0,C 180,E1 -1168.644,E2 -1168.644} C_VEL
LIN {X 0,Y 594.233,Z 710.5,A -85,B 0,C 180,E1 -1170,E2 -1170} C_VEL
LIN {X 0,Y 594.245,Z 709.913,A -85,B 0,C 180,E1 -1171.355,E2 -1171.355} C_VEL
LIN {X 0,Y 594.223,Z 708.186,A -85,B 0,C 180,E1 -1172.711,E2 -1172.711} C_VEL
LIN {X 0,Y 594.253,Z 705.289,A -85,B 0,C 180,E1 -1174.069,E2 -1174.069} C_VEL
LIN {X 0,Y 594.273,Z 701.163,A -85,B 0,C 180,E1 -1175.428,E2 -1175.428} C_VEL
LIN {X 0,Y 594.274,Z 695.705,A -85,B 0,C 180,E1 -1176.791,E2 -1176.791} C_VEL
LIN {X 0,Y 594.323,Z 688.754,A -85,B 0,C 180,E1 -1178.157,E2 -1178.157} C_VEL
LIN {X 0,Y 594.341,Z 680.096,A -85,B 0,C 180,E1 -1179.529,E2 -1179.529} C_VEL
LIN {X 0,Y 594.401,Z 670.882,A -85,B 0,C 180,E1 -1180.732,E2 -1180.732} C_VEL
LIN {X 0,Y 594.467,Z 661.514,A -85,B 0,C 180,E1 -1181.767,E2 -1181.767} C_VEL
LIN {X 0,Y 594.551,Z 650.395,A -85,B 0,C 180,E1 -1182.805,E2 -1182.805} C_VEL
LIN {X 0,Y 594.652,Z 637.655,A -85,B 0,C 180,E1 -1183.798,E2 -1183.798} C_VEL
LIN {X 0,Y 594.744,Z 624.793,A -85,B 0,C 180,E1 -1184.63,E2 -1184.63} C_VEL
LIN {X 0,Y 594.816,Z 611.622,A -85,B 0,C 180,E1 -1185.329,E2 -1185.329} C_VEL
LIN {X 0,Y 594.907,Z 597.2,A -85,B 0,C 180,E1 -1185.941,E2 -1185.941} C_VEL
LIN {X 0,Y 595.005,Z 582.276,A -85,B 0,C 180,E1 -1186.423,E2 -1186.423} C_VEL
LIN {X 0,Y 595.094,Z 567.29,A -85,B 0,C 180,E1 -1186.764,E2 -1186.764} C_VEL
LIN {X 0,Y 594.902,Z 557.081,A -85,B 0,C 180,E1 -1186.928,E2 -1186.928} C_VEL
LIN {X 0,Y 594.328,Z 554.412,A -85,B 0,C 180,E1 -1186.983,E2 -1186.983} C_VEL
LIN {X 0,Y 594.371,Z 545.01,A -85,B 0,C 180,E1 -1189.693,E2 -1189.693} C_VEL
LIN {X 0,Y 594.406,Z 536.346,A -85,B 0,C 180,E1 -1192.231,E2 -1192.231} C_VEL
LIN {X 0,Y 594.432,Z 527.681,A -85,B 0,C 180,E1 -1194.816,E2 -1194.816} C_VEL
LIN {X 0,Y 594.473,Z 518.732,A -85,B 0,C 180,E1 -1197.543,E2 -1197.543} C_VEL
LIN {X 0,Y 594.514,Z 509.75,A -85,B 0,C 180,E1 -1200.349,E2 -1200.349} C_VEL
LIN {X 0,Y 594.556,Z 501.688,A -85,B 0,C 180,E1 -1202.938,E2 -1202.938} C_VEL
LIN {X 0,Y 594.587,Z 492.756,A -85,B 0,C 180,E1 -1205.808,E2 -1205.808} C_VEL
LIN {X 0,Y 594.644,Z 484.033,A -85,B 0,C 180,E1 -1208.784,E2 -1208.784} C_VEL
LIN {X 0,Y 594.64,Z 476.659,A -85,B 0,C 180,E1 -1211.44,E2 -1211.44} C_VEL
LIN {X 0,Y 594.405,Z 475.073,A -85,B 0,C 180,E1 -1212.081,E2 -1212.081} C_VEL
LIN {X 0,Y 594.356,Z 475.076,A -85,B 0,C 180,E1 -1214.808,E2 -1214.808} C_VEL
LIN {X 0,Y 594.383,Z 475.076,A -85,B 0,C 180,E1 -1217.626,E2 -1217.626} C_VEL
LIN {X 0,Y 594.394,Z 475.071,A -85,B 0,C 180,E1 -1220.321,E2 -1220.321} C_VEL
LIN {X 0,Y 594.38,Z 475.074,A -85,B 0,C 180,E1 -1222.913,E2 -1222.913} C_VEL
LIN {X 0,Y 594.382,Z 475.073,A -85,B 0,C 180,E1 -1225.859,E2 -1225.859} C_VEL
LIN {X 0,Y 594.385,Z 475.075,A -85,B 0,C 180,E1 -1228.651,E2 -1228.651} C_VEL
LIN {X 0,Y 594.382,Z 475.074,A -85,B 0,C 180,E1 -1231.04,E2 -1231.04} C_VEL
LIN {X 0,Y 594.388,Z 475.074,A -85,B 0,C 180,E1 -1233.974,E2 -1233.974} C_VEL
LIN {X 0,Y 594.384,Z 475.075,A -85,B 0,C 180,E1 -1236.296,E2 -1236.296} C_VEL
LIN {X 0,Y 594.404,Z 475.07,A -85,B 0,C 180,E1 -1239.225,E2 -1239.225} C_VEL
LIN {X 0,Y 594.375,Z 475.074,A -85,B 0,C 180,E1 -1242.096,E2 -1242.096} C_VEL
LIN {X 0,Y 594.367,Z 475.076,A -85,B 0,C 180,E1 -1244.219,E2 -1244.219} C_VEL
LIN {X 0,Y 594.366,Z 475.075,A -85,B 0,C 180,E1 -1247.017,E2 -1247.017} C_VEL
LIN {X 0,Y 594.391,Z 475.073,A -85,B 0,C 180,E1 -1249.784,E2 -1249.784} C_VEL
LIN {X 0,Y 594.413,Z 475.069,A -85,B 0,C 180,E1 -1252.527,E2 -1252.527} C_VEL
LIN {X 0,Y 594.396,Z 475.073,A -85,B 0,C 180,E1 -1255.253,E2 -1255.253} C_VEL
LIN {X 0,Y 594.391,Z 475.072,A -85,B 0,C 180,E1 -1257.967,E2 -1257.967} C_VEL
LIN {X 0,Y 594.421,Z 475.07,A -85,B 0,C 180,E1 -1260.678,E2 -1260.678} C_VEL
LIN {X 0,Y 594.383,Z 475.073,A -85,B 0,C 180,E1 -1263.39,E2 -1263.39} C_VEL
LIN {X 0,Y 594.39,Z 475.074,A -85,B 0,C 180,E1 -1266.109,E2 -1266.109} C_VEL
LIN {X 0,Y 594.396,Z 475.071,A -85,B 0,C 180,E1 -1268.842,E2 -1268.842} C_VEL
LIN {X 0,Y 594.385,Z 475.075,A -85,B 0,C 180,E1 -1271.596,E2 -1271.596} C_VEL
LIN {X 0,Y 594.381,Z 475.073,A -85,B 0,C 180,E1 -1274.378,E2 -1274.378} C_VEL
LIN {X 0,Y 594.362,Z 475.075,A -85,B 0,C 180,E1 -1275.341,E2 -1275.341} C_VEL
LIN {X 0,Y 593.694,Z 475.161,A -85,B 0,C 180,E1 -1275.907,E2 -1275.907} C_VEL
LIN {X 0,Y 590.841,Z 475.517,A -85,B 0,C 180,E1 -1276.825,E2 -1276.825} C_VEL
LIN {X 0,Y 588.434,Z 475.817,A -85,B 0,C 180,E1 -1277.564,E2 -1277.564} C_VEL
LIN {X 0,Y 587.405,Z 475.944,A -85,B 0,C 180,E1 -1278.134,E2 -1278.134} C_VEL
LIN {X 0,Y 587.324,Z 475.953,A -85,B 0,C 180,E1 -1278.327,E2 -1278.327} C_VEL
LIN {X 0,Y 587.349,Z 475.949,A -85,B 0,C 180,E1 -1281.046,E2 -1281.046} C_VEL
LIN {X 0,Y 587.331,Z 475.951,A -85,B 0,C 180,E1 -1284.007,E2 -1284.007} C_VEL
LIN {X 0,Y 587.359,Z 475.947,A -85,B 0,C 180,E1 -1286.278,E2 -1286.278} C_VEL
LIN {X 0,Y 587.348,Z 475.951,A -85,B 0,C 180,E1 -1289.136,E2 -1289.136} C_VEL
LIN {X 0,Y 587.353,Z 475.948,A -85,B 0,C 180,E1 -1291.839,E2 -1291.839} C_VEL
LIN {X 0,Y 587.353,Z 475.949,A -85,B 0,C 180,E1 -1294.351,E2 -1294.351} C_VEL
LIN {X 0,Y 587.349,Z 475.95,A -85,B 0,C 180,E1 -1296.747,E2 -1296.747} C_VEL
LIN {X 0,Y 587.346,Z 475.95,A -85,B 0,C 180,E1 -1299.36,E2 -1299.36} C_VEL
LIN {X 0,Y 587.33,Z 475.952,A -85,B 0,C 180,E1 -1302.109,E2 -1302.109} C_VEL
LIN {X 0,Y 587.312,Z 475.953,A -85,B 0,C 180,E1 -1305.09,E2 -1305.09} C_VEL
LIN {X 0,Y 587.35,Z 475.952,A -85,B 0,C 180,E1 -1307.929,E2 -1307.929} C_VEL
LIN {X 0,Y 587.346,Z 475.949,A -85,B 0,C 180,E1 -1310.642,E2 -1310.642} C_VEL
LIN {X 0,Y 587.354,Z 475.95,A -85,B 0,C 180,E1 -1313.293,E2 -1313.293} C_VEL
LIN {X 0,Y 587.361,Z 475.949,A -85,B 0,C 180,E1 -1315.781,E2 -1315.781} C_VEL
LIN {X 0,Y 587.352,Z 475.948,A -85,B 0,C 180,E1 -1318.233,E2 -1318.233} C_VEL
LIN {X 0,Y 587.351,Z 475.949,A -85,B 0,C 180,E1 -1320.867,E2 -1320.867} C_VEL
LIN {X 0,Y 587.364,Z 475.947,A -85,B 0,C 180,E1 -1323.819,E2 -1323.819} C_VEL
LIN {X 0,Y 587.341,Z 475.95,A -85,B 0,C 180,E1 -1325.995,E2 -1325.995} C_VEL
LIN {X 0,Y 587.324,Z 475.952,A -85,B 0,C 180,E1 -1328.227,E2 -1328.227} C_VEL
LIN {X 0,Y 587.352,Z 475.951,A -85,B 0,C 180,E1 -1331.152,E2 -1331.152} C_VEL
LIN {X 0,Y 587.355,Z 475.951,A -85,B 0,C 180,E1 -1333.312,E2 -1333.312} C_VEL
LIN {X 0,Y 587.364,Z 475.947,A -85,B 0,C 180,E1 -1336.155,E2 -1336.155} C_VEL
LIN {X 0,Y 587.344,Z 475.951,A -85,B 0,C 180,E1 -1338.963,E2 -1338.963} C_VEL
LIN {X 0,Y 587.346,Z 475.95,A -85,B 0,C 180,E1 -1341.745,E2 -1341.745} C_VEL
LIN {X 0,Y 587.36,Z 475.948,A -85,B 0,C 180,E1 -1344.508,E2 -1344.508} C_VEL
LIN {X 0,Y 587.375,Z 475.946,A -85,B 0,C 180,E1 -1347.257,E2 -1347.257} C_VEL
LIN {X 0,Y 587.389,Z 475.945,A -85,B 0,C 180,E1 -1350,E2 -1350} C_VEL
LIN {X 0,Y 587.365,Z 475.95,A -85,B 0,C 180,E1 -1352.057,E2 -1352.057} C_VEL
LIN {X 0,Y 587.224,Z 475.968,A -85,B 0,C 180,E1 -1352.744,E2 -1352.744} C_VEL
LIN {X 0,Y 587.26,Z 477.954,A -85,B 0,C 180,E1 -1354.806,E2 -1354.806} C_VEL
LIN {X 0,Y 587.224,Z 480.768,A -85,B 0,C 180,E1 -1357.565,E2 -1357.565} C_VEL
LIN {X 0,Y 587.158,Z 483.644,A -85,B 0,C 180,E1 -1360.343,E2 -1360.343} C_VEL
LIN {X 0,Y 587.176,Z 486.805,A -85,B 0,C 180,E1 -1363.145,E2 -1363.145} C_VEL
LIN {X 0,Y 587.17,Z 489.254,A -85,B 0,C 180,E1 -1365.267,E2 -1365.267} C_VEL
LIN {X 0,Y 587.13,Z 491.774,A -85,B 0,C 180,E1 -1367.413,E2 -1367.413} C_VEL
LIN {X 0,Y 587.133,Z 494.36,A -85,B 0,C 180,E1 -1369.582,E2 -1369.582} C_VEL
LIN {X 0,Y 587.149,Z 497.922,A -85,B 0,C 180,E1 -1372.521,E2 -1372.521} C_VEL
LIN {X 0,Y 587.155,Z 498.409,A -85,B 0,C 180,E1 -1372.905,E2 -1372.905} C_VEL
LIN {X 0,Y 588.267,Z 504.244,A -85,B 0,C 180,E1 -1373.025,E2 -1373.025} C_VEL
LIN {X 0,Y 588.217,Z 520.383,A -85,B 0,C 180,E1 -1373.373,E2 -1373.373} C_VEL
LIN {X 0,Y 588.084,Z 535.079,A -85,B 0,C 180,E1 -1373.834,E2 -1373.834} C_VEL
LIN {X 0,Y 587.991,Z 549.809,A -85,B 0,C 180,E1 -1374.446,E2 -1374.446} C_VEL
LIN {X 0,Y 587.816,Z 562.63,A -85,B 0,C 180,E1 -1375.115,E2 -1375.115} C_VEL
LIN {X 0,Y 587.703,Z 576.042,A -85,B 0,C 180,E1 -1375.968,E2 -1375.968} C_VEL
LIN {X 0,Y 587.577,Z 588.629,A -85,B 0,C 180,E1 -1376.938,E2 -1376.938} C_VEL
LIN {X 0,Y 587.45,Z 600.217,A -85,B 0,C 180,E1 -1378.006,E2 -1378.006} C_VEL
LIN {X 0,Y 587.364,Z 610.471,A -85,B 0,C 180,E1 -1379.135,E2 -1379.135} C_VEL
LIN {X 0,Y 587.304,Z 619.627,A -85,B 0,C 180,E1 -1380.335,E2 -1380.335} C_VEL
LIN {X 0,Y 587.243,Z 627.499,A -85,B 0,C 180,E1 -1381.573,E2 -1381.573} C_VEL
LIN {X 0,Y 587.184,Z 634.142,A -85,B 0,C 180,E1 -1382.837,E2 -1382.837} C_VEL
LIN {X 0,Y 587.164,Z 640.023,A -85,B 0,C 180,E1 -1384.233,E2 -1384.233} C_VEL
LIN {X 0,Y 587.15,Z 644.227,A -85,B 0,C 180,E1 -1385.517,E2 -1385.517} C_VEL
LIN {X 0,Y 587.124,Z 647.198,A -85,B 0,C 180,E1 -1386.763,E2 -1386.763} C_VEL
LIN {X 0,Y 587.119,Z 648.986,A -85,B 0,C 180,E1 -1387.81,E2 -1387.81} C_VEL
LIN {X 0,Y 587.11,Z 650.354,A -85,B 0,C 180,E1 -1389.378,E2 -1389.378} C_VEL
LIN {X 0,Y 587.136,Z 650.455,A -85,B 0,C 180,E1 -1390.269,E2 -1390.269} C_VEL
LIN {X 0,Y 587.121,Z 650.078,A -85,B 0,C 180,E1 -1391.175,E2 -1391.175} C_VEL
LIN {X 0,Y 587.165,Z 649.209,A -85,B 0,C 180,E1 -1392.089,E2 -1392.089} C_VEL
LIN {X 0,Y 587.147,Z 647.67,A -85,B 0,C 180,E1 -1393.1,E2 -1393.1} C_VEL
LIN {X 0,Y 587.169,Z 644.459,A -85,B 0,C 180,E1 -1394.485,E2 -1394.485} C_VEL
LIN {X 0,Y 587.182,Z 639.379,A -85,B 0,C 180,E1 -1396.036,E2 -1396.036} C_VEL
LIN {X 0,Y 587.218,Z 633.211,A -85,B 0,C 180,E1 -1397.452,E2 -1397.452} C_VEL
LIN {X 0,Y 587.23,Z 625.654,A -85,B 0,C 180,E1 -1398.833,E2 -1398.833} C_VEL
LIN {X 0,Y 587.307,Z 616.857,A -85,B 0,C 180,E1 -1400.144,E2 -1400.144} C_VEL
LIN {X 0,Y 587.415,Z 606.58,A -85,B 0,C 180,E1 -1401.41,E2 -1401.41} C_VEL
LIN {X 0,Y 587.486,Z 595.87,A -85,B 0,C 180,E1 -1402.511,E2 -1402.511} C_VEL
LIN {X 0,Y 587.614,Z 584.596,A -85,B 0,C 180,E1 -1403.485,E2 -1403.485} C_VEL
LIN {X 0,Y 587.751,Z 571.988,A -85,B 0,C 180,E1 -1404.4,E2 -1404.4} C_VEL
LIN {X 0,Y 587.879,Z 558.036,A -85,B 0,C 180,E1 -1405.232,E2 -1405.232} C_VEL
LIN {X 0,Y 588.022,Z 543.502,A -85,B 0,C 180,E1 -1405.927,E2 -1405.927} C_VEL
LIN {X 0,Y 588.152,Z 529.392,A -85,B 0,C 180,E1 -1406.45,E2 -1406.45} C_VEL
LIN {X 0,Y 588.229,Z 514.203,A -85,B 0,C 180,E1 -1406.868,E2 -1406.868} C_VEL
LIN {X 0,Y 588.192,Z 503.143,A -85,B 0,C 180,E1 -1407.084,E2 -1407.084} C_VEL
LIN {X 0,Y 587.161,Z 498.372,A -85,B 0,C 180,E1 -1407.2,E2 -1407.2} C_VEL
LIN {X 0,Y 587.156,Z 495.188,A -85,B 0,C 180,E1 -1409.819,E2 -1409.819} C_VEL
LIN {X 0,Y 587.165,Z 492.171,A -85,B 0,C 180,E1 -1412.341,E2 -1412.341} C_VEL
LIN {X 0,Y 587.175,Z 488.777,A -85,B 0,C 180,E1 -1415.233,E2 -1415.233} C_VEL
LIN {X 0,Y 587.166,Z 485.357,A -85,B 0,C 180,E1 -1418.219,E2 -1418.219} C_VEL
LIN {X 0,Y 587.222,Z 482.092,A -85,B 0,C 180,E1 -1421.147,E2 -1421.147} C_VEL
LIN {X 0,Y 587.274,Z 480.242,A -85,B 0,C 180,E1 -1423.309,E2 -1423.309} C_VEL
LIN {X 0,Y 587.243,Z 477.351,A -85,B 0,C 180,E1 -1426.151,E2 -1426.151} C_VEL
LIN {X 0,Y 587.256,Z 475.963,A -85,B 0,C 180,E1 -1427.56,E2 -1427.56} C_VEL
LIN {X 0,Y 587.345,Z 475.946,A -85,B 0,C 180,E1 -1429.66,E2 -1429.66} C_VEL
LIN {X 0,Y 587.364,Z 475.944,A -85,B 0,C 180,E1 -1432.437,E2 -1432.437} C_VEL
LIN {X 0,Y 587.367,Z 475.941,A -85,B 0,C 180,E1 -1435.195,E2 -1435.195} C_VEL
LIN {X 0,Y 587.366,Z 475.946,A -85,B 0,C 180,E1 -1437.943,E2 -1437.943} C_VEL
LIN {X 0,Y 587.391,Z 475.937,A -85,B 0,C 180,E1 -1440.685,E2 -1440.685} C_VEL
LIN {X 0,Y 587.33,Z 475.954,A -85,B 0,C 180,E1 -1443.43,E2 -1443.43} C_VEL
LIN {X 0,Y 587.36,Z 475.948,A -85,B 0,C 180,E1 -1445.493,E2 -1445.493} C_VEL
LIN {X 0,Y 587.367,Z 475.94,A -85,B 0,C 180,E1 -1448.255,E2 -1448.255} C_VEL
LIN {X 0,Y 587.358,Z 475.949,A -85,B 0,C 180,E1 -1451.141,E2 -1451.141} C_VEL
LIN {X 0,Y 587.36,Z 475.943,A -85,B 0,C 180,E1 -1454.26,E2 -1454.26} C_VEL
LIN {X 0,Y 587.347,Z 475.943,A -85,B 0,C 180,E1 -1457.406,E2 -1457.406} C_VEL
LIN {X 0,Y 587.329,Z 475.951,A -85,B 0,C 180,E1 -1460.305,E2 -1460.305} C_VEL
LIN {X 0,Y 587.319,Z 475.946,A -85,B 0,C 180,E1 -1463.259,E2 -1463.259} C_VEL
LIN {X 0,Y 587.337,Z 475.945,A -85,B 0,C 180,E1 -1465.516,E2 -1465.516} C_VEL
LIN {X 0,Y 587.346,Z 475.948,A -85,B 0,C 180,E1 -1467.818,E2 -1467.818} C_VEL
LIN {X 0,Y 587.347,Z 475.945,A -85,B 0,C 180,E1 -1470.513,E2 -1470.513} C_VEL
LIN {X 0,Y 587.332,Z 475.948,A -85,B 0,C 180,E1 -1473.397,E2 -1473.397} C_VEL
LIN {X 0,Y 587.354,Z 475.949,A -85,B 0,C 180,E1 -1475.895,E2 -1475.895} C_VEL
LIN {X 0,Y 587.329,Z 475.945,A -85,B 0,C 180,E1 -1478.479,E2 -1478.479} C_VEL
LIN {X 0,Y 587.335,Z 475.95,A -85,B 0,C 180,E1 -1481.157,E2 -1481.157} C_VEL
LIN {X 0,Y 587.332,Z 475.946,A -85,B 0,C 180,E1 -1484.114,E2 -1484.114} C_VEL
LIN {X 0,Y 587.335,Z 475.953,A -85,B 0,C 180,E1 -1486.996,E2 -1486.996} C_VEL
LIN {X 0,Y 587.356,Z 476.13,A -85,B 0,C 180,E1 -1487.813,E2 -1487.813} C_VEL
LIN {X 0,Y 587.702,Z 480.051,A -85,B 0,C 180,E1 -1489.334,E2 -1489.334} C_VEL
LIN {X 0,Y 587.637,Z 486.202,A -85,B 0,C 180,E1 -1491.545,E2 -1491.545} C_VEL
LIN {X 0,Y 587.582,Z 494.588,A -85,B 0,C 180,E1 -1494.423,E2 -1494.423} C_VEL
LIN {X 0,Y 587.556,Z 502.238,A -85,B 0,C 180,E1 -1496.856,E2 -1496.856} C_VEL
LIN {X 0,Y 587.551,Z 510.379,A -85,B 0,C 180,E1 -1499.455,E2 -1499.455} C_VEL
LIN {X 0,Y 587.472,Z 519.32,A -85,B 0,C 180,E1 -1502.285,E2 -1502.285} C_VEL
LIN {X 0,Y 587.414,Z 527.679,A -85,B 0,C 180,E1 -1504.866,E2 -1504.866} C_VEL
LIN {X 0,Y 587.364,Z 536.343,A -85,B 0,C 180,E1 -1507.487,E2 -1507.487} C_VEL
LIN {X 0,Y 587.321,Z 546.245,A -85,B 0,C 180,E1 -1510.424,E2 -1510.424} C_VEL
LIN {X 0,Y 587.266,Z 554.425,A -85,B 0,C 180,E1 -1512.81,E2 -1512.81} C_VEL
LIN {X 0,Y 588.295,Z 559.894,A -85,B 0,C 180,E1 -1512.916,E2 -1512.916} C_VEL
LIN {X 0,Y 588.233,Z 575.344,A -85,B 0,C 180,E1 -1513.205,E2 -1513.205} C_VEL
LIN {X 0,Y 588.14,Z 589.611,A -85,B 0,C 180,E1 -1513.602,E2 -1513.602} C_VEL
LIN {X 0,Y 588.053,Z 603.838,A -85,B 0,C 180,E1 -1514.134,E2 -1514.134} C_VEL
LIN {X 0,Y 587.885,Z 618.524,A -85,B 0,C 180,E1 -1514.84,E2 -1514.84} C_VEL
LIN {X 0,Y 587.757,Z 631.163,A -85,B 0,C 180,E1 -1515.59,E2 -1515.59} C_VEL
LIN {X 0,Y 587.629,Z 644.013,A -85,B 0,C 180,E1 -1516.513,E2 -1516.513} C_VEL
LIN {X 0,Y 587.522,Z 656.19,A -85,B 0,C 180,E1 -1517.566,E2 -1517.566} C_VEL
LIN {X 0,Y 587.424,Z 666.704,A -85,B 0,C 180,E1 -1518.649,E2 -1518.649} C_VEL
LIN {X 0,Y 587.351,Z 676.369,A -85,B 0,C 180,E1 -1519.834,E2 -1519.834} C_VEL
LIN {X 0,Y 587.267,Z 684.652,A -85,B 0,C 180,E1 -1521.05,E2 -1521.05} C_VEL
LIN {X 0,Y 587.23,Z 692.424,A -85,B 0,C 180,E1 -1522.435,E2 -1522.435} C_VEL
LIN {X 0,Y 587.178,Z 698.606,A -85,B 0,C 180,E1 -1523.816,E2 -1523.816} C_VEL
LIN {X 0,Y 587.136,Z 703.383,A -85,B 0,C 180,E1 -1525.193,E2 -1525.193} C_VEL
LIN {X 0,Y 587.179,Z 706.887,A -85,B 0,C 180,E1 -1526.569,E2 -1526.569} C_VEL
LIN {X 0,Y 587.137,Z 709.193,A -85,B 0,C 180,E1 -1527.942,E2 -1527.942} C_VEL
LIN {X 0,Y 587.137,Z 710.35,A -85,B 0,C 180,E1 -1529.314,E2 -1529.314} C_VEL
LIN {X 0,Y 587.137,Z 710.35,A -85,B 0,C 180,E1 -1530.685,E2 -1530.685} C_VEL
LIN {X 0,Y 587.137,Z 709.193,A -85,B 0,C 180,E1 -1532.058,E2 -1532.058} C_VEL
LIN {X 0,Y 587.179,Z 706.887,A -85,B 0,C 180,E1 -1533.431,E2 -1533.431} C_VEL
LIN {X 0,Y 587.136,Z 703.385,A -85,B 0,C 180,E1 -1534.806,E2 -1534.806} C_VEL
LIN {X 0,Y 587.178,Z 698.61,A -85,B 0,C 180,E1 -1536.184,E2 -1536.184} C_VEL
LIN {X 0,Y 587.235,Z 692.427,A -85,B 0,C 180,E1 -1537.564,E2 -1537.564} C_VEL
LIN {X 0,Y 587.266,Z 684.655,A -85,B 0,C 180,E1 -1538.95,E2 -1538.95} C_VEL
LIN {X 0,Y 587.351,Z 676.374,A -85,B 0,C 180,E1 -1540.165,E2 -1540.165} C_VEL
LIN {X 0,Y 587.399,Z 666.4,A -85,B 0,C 180,E1 -1541.385,E2 -1541.385} C_VEL
LIN {X 0,Y 587.521,Z 656.197,A -85,B 0,C 180,E1 -1542.434,E2 -1542.434} C_VEL
LIN {X 0,Y 587.628,Z 644.025,A -85,B 0,C 180,E1 -1543.486,E2 -1543.486} C_VEL
LIN {X 0,Y 587.773,Z 631.064,A -85,B 0,C 180,E1 -1544.416,E2 -1544.416} C_VEL
LIN {X 0,Y 587.886,Z 616.876,A -85,B 0,C 180,E1 -1545.248,E2 -1545.248} C_VEL
LIN {X 0,Y 588.049,Z 602.811,A -85,B 0,C 180,E1 -1545.91,E2 -1545.91} C_VEL
LIN {X 0,Y 588.165,Z 588.323,A -85,B 0,C 180,E1 -1546.441,E2 -1546.441} C_VEL
LIN {X 0,Y 588.282,Z 572.734,A -85,B 0,C 180,E1 -1546.857,E2 -1546.857} C_VEL
LIN {X 0,Y 588.253,Z 558.682,A -85,B 0,C 180,E1 -1547.103,E2 -1547.103} C_VEL
LIN {X 0,Y 587.268,Z 554.375,A -85,B 0,C 180,E1 -1547.205,E2 -1547.205} C_VEL
LIN {X 0,Y 587.327,Z 545.01,A -85,B 0,C 180,E1 -1549.939,E2 -1549.939} C_VEL
LIN {X 0,Y 587.362,Z 536.346,A -85,B 0,C 180,E1 -1552.512,E2 -1552.512} C_VEL
LIN {X 0,Y 587.441,Z 526.443,A -85,B 0,C 180,E1 -1555.511,E2 -1555.511} C_VEL
LIN {X 0,Y 587.495,Z 517.779,A -85,B 0,C 180,E1 -1558.197,E2 -1558.197} C_VEL
LIN {X 0,Y 587.544,Z 509.114,A -85,B 0,C 180,E1 -1560.953,E2 -1560.953} C_VEL
LIN {X 0,Y 587.588,Z 500.297,A -85,B 0,C 180,E1 -1563.791,E2 -1563.791} C_VEL
LIN {X 0,Y 587.584,Z 492.602,A -85,B 0,C 180,E1 -1566.302,E2 -1566.302} C_VEL
LIN {X 0,Y 587.7,Z 484.918,A -85,B 0,C 180,E1 -1568.986,E2 -1568.986} C_VEL
LIN {X 0,Y 587.721,Z 479.041,A -85,B 0,C 180,E1 -1571.123,E2 -1571.123} C_VEL
LIN {X 0,Y 587.348,Z 475.951,A -85,B 0,C 180,E1 -1572.36,E2 -1572.36} C_VEL
LIN {X 0,Y 587.308,Z 475.955,A -85,B 0,C 180,E1 -1575.088,E2 -1575.088} C_VEL
LIN {X 0,Y 587.345,Z 475.95,A -85,B 0,C 180,E1 -1577.927,E2 -1577.927} C_VEL
LIN {X 0,Y 587.346,Z 475.95,A -85,B 0,C 180,E1 -1580.641,E2 -1580.641} C_VEL
LIN {X 0,Y 587.346,Z 475.951,A -85,B 0,C 180,E1 -1583.291,E2 -1583.291} C_VEL
LIN {X 0,Y 587.364,Z 475.947,A -85,B 0,C 180,E1 -1585.78,E2 -1585.78} C_VEL
LIN {X 0,Y 587.349,Z 475.949,A -85,B 0,C 180,E1 -1588.232,E2 -1588.232} C_VEL
LIN {X 0,Y 587.347,Z 475.952,A -85,B 0,C 180,E1 -1590.865,E2 -1590.865} C_VEL
LIN {X 0,Y 587.356,Z 475.949,A -85,B 0,C 180,E1 -1593.817,E2 -1593.817} C_VEL
LIN {X 0,Y 587.315,Z 475.953,A -85,B 0,C 180,E1 -1596.741,E2 -1596.741} C_VEL
LIN {X 0,Y 587.33,Z 475.954,A -85,B 0,C 180,E1 -1599.695,E2 -1599.695} C_VEL
LIN {X 0,Y 587.351,Z 475.948,A -85,B 0,C 180,E1 -1602.594,E2 -1602.594} C_VEL
LIN {X 0,Y 587.354,Z 475.948,A -85,B 0,C 180,E1 -1605.739,E2 -1605.739} C_VEL
LIN {X 0,Y 587.351,Z 475.949,A -85,B 0,C 180,E1 -1608.859,E2 -1608.859} C_VEL
LIN {X 0,Y 587.366,Z 475.95,A -85,B 0,C 180,E1 -1611.745,E2 -1611.745} C_VEL
LIN {X 0,Y 587.356,Z 475.947,A -85,B 0,C 180,E1 -1614.507,E2 -1614.507} C_VEL
LIN {X 0,Y 587.377,Z 475.948,A -85,B 0,C 180,E1 -1617.257,E2 -1617.257} C_VEL
LIN {X 0,Y 587.373,Z 475.946,A -85,B 0,C 180,E1 -1620,E2 -1620} C_VEL
LIN {X 0,Y 587.377,Z 475.948,A -85,B 0,C 180,E1 -1622.744,E2 -1622.744} C_VEL
LIN {X 0,Y 587.365,Z 475.947,A -85,B 0,C 180,E1 -1625.493,E2 -1625.493} C_VEL
LIN {X 0,Y 587.366,Z 475.949,A -85,B 0,C 180,E1 -1628.256,E2 -1628.256} C_VEL
LIN {X 0,Y 587.352,Z 475.948,A -85,B 0,C 180,E1 -1631.142,E2 -1631.142} C_VEL
LIN {X 0,Y 587.355,Z 475.948,A -85,B 0,C 180,E1 -1634.262,E2 -1634.262} C_VEL
LIN {X 0,Y 587.355,Z 475.949,A -85,B 0,C 180,E1 -1637.406,E2 -1637.406} C_VEL
LIN {X 0,Y 587.324,Z 475.953,A -85,B 0,C 180,E1 -1638.327,E2 -1638.327} C_VEL
LIN {X 0,Y 586.669,Z 476.034,A -85,B 0,C 180,E1 -1638.899,E2 -1638.899} C_VEL
LIN {X 0,Y 583.837,Z 476.388,A -85,B 0,C 180,E1 -1639.827,E2 -1639.827} C_VEL
LIN {X 0,Y 581.427,Z 476.69,A -85,B 0,C 180,E1 -1640.574,E2 -1640.574} C_VEL
LIN {X 0,Y 580.374,Z 476.82,A -85,B 0,C 180,E1 -1641.151,E2 -1641.151} C_VEL
LIN {X 0,Y 580.279,Z 476.83,A -85,B 0,C 180,E1 -1641.346,E2 -1641.346} C_VEL
LIN {X 0,Y 580.294,Z 476.827,A -85,B 0,C 180,E1 -1644.317,E2 -1644.317} C_VEL
LIN {X 0,Y 580.308,Z 476.826,A -85,B 0,C 180,E1 -1646.622,E2 -1646.622} C_VEL
LIN {X 0,Y 580.302,Z 476.829,A -85,B 0,C 180,E1 -1649.312,E2 -1649.312} C_VEL
LIN {X 0,Y 580.299,Z 476.828,A -85,B 0,C 180,E1 -1652.201,E2 -1652.201} C_VEL
LIN {X 0,Y 580.297,Z 476.829,A -85,B 0,C 180,E1 -1654.696,E2 -1654.696} C_VEL
LIN {X 0,Y 580.297,Z 476.828,A -85,B 0,C 180,E1 -1657.269,E2 -1657.269} C_VEL
LIN {X 0,Y 580.304,Z 476.828,A -85,B 0,C 180,E1 -1660.274,E2 -1660.274} C_VEL
LIN {X 0,Y 580.278,Z 476.83,A -85,B 0,C 180,E1 -1662.707,E2 -1662.707} C_VEL
LIN {X 0,Y 580.271,Z 476.833,A -85,B 0,C 180,E1 -1665.61,E2 -1665.61} C_VEL
LIN {X 0,Y 580.303,Z 476.826,A -85,B 0,C 180,E1 -1668.667,E2 -1668.667} C_VEL
LIN {X 0,Y 580.29,Z 476.828,A -85,B 0,C 180,E1 -1670.967,E2 -1670.967} C_VEL
LIN {X 0,Y 580.293,Z 476.829,A -85,B 0,C 180,E1 -1673.599,E2 -1673.599} C_VEL
LIN {X 0,Y 580.303,Z 476.829,A -85,B 0,C 180,E1 -1676.685,E2 -1676.685} C_VEL
LIN {X 0,Y 580.304,Z 476.826,A -85,B 0,C 180,E1 -1679.427,E2 -1679.427} C_VEL
LIN {X 0,Y 580.322,Z 476.826,A -85,B 0,C 180,E1 -1682.138,E2 -1682.138} C_VEL
LIN {X 0,Y 580.312,Z 476.825,A -85,B 0,C 180,E1 -1684.921,E2 -1684.921} C_VEL
LIN {X 0,Y 580.275,Z 476.831,A -85,B 0,C 180,E1 -1687.948,E2 -1687.948} C_VEL
LIN {X 0,Y 580.301,Z 476.828,A -85,B 0,C 180,E1 -1690.914,E2 -1690.914} C_VEL
LIN {X 0,Y 580.315,Z 476.826,A -85,B 0,C 180,E1 -1693.103,E2 -1693.103} C_VEL
LIN {X 0,Y 580.331,Z 476.823,A -85,B 0,C 180,E1 -1695.984,E2 -1695.984} C_VEL
LIN {X 0,Y 580.31,Z 476.828,A -85,B 0,C 180,E1 -1698.828,E2 -1698.828} C_VEL
LIN {X 0,Y 580.315,Z 476.825,A -85,B 0,C 180,E1 -1701.644,E2 -1701.644} C_VEL
LIN {X 0,Y 580.289,Z 476.828,A -85,B 0,C 180,E1 -1703.743,E2 -1703.743} C_VEL
LIN {X 0,Y 580.279,Z 476.83,A -85,B 0,C 180,E1 -1705.833,E2 -1705.833} C_VEL
LIN {X 0,Y 580.345,Z 476.822,A -85,B 0,C 180,E1 -1707.918,E2 -1707.918} C_VEL
LIN {X 0,Y 580.366,Z 476.82,A -85,B 0,C 180,E1 -1710.694,E2 -1710.694} C_VEL
LIN {X 0,Y 580.173,Z 476.846,A -85,B 0,C 180,E1 -1712.778,E2 -1712.778} C_VEL
LIN {X 0,Y 580.2,Z 478.634,A -85,B 0,C 180,E1 -1714.864,E2 -1714.864} C_VEL
LIN {X 0,Y 580.147,Z 480.706,A -85,B 0,C 180,E1 -1716.958,E2 -1716.958} C_VEL
LIN {X 0,Y 580.101,Z 482.816,A -85,B 0,C 180,E1 -1719.062,E2 -1719.062} C_VEL
LIN {X 0,Y 580.103,Z 485.791,A -85,B 0,C 180,E1 -1721.886,E2 -1721.886} C_VEL
LIN {X 0,Y 580.112,Z 489.018,A -85,B 0,C 180,E1 -1724.739,E2 -1724.739} C_VEL
LIN {X 0,Y 580.068,Z 491.521,A -85,B 0,C 180,E1 -1726.905,E2 -1726.905} C_VEL
LIN {X 0,Y 580.057,Z 494.965,A -85,B 0,C 180,E1 -1729.831,E2 -1729.831} C_VEL
LIN {X 0,Y 580.051,Z 498.37,A -85,B 0,C 180,E1 -1732.671,E2 -1732.671} C_VEL
LIN {X 0,Y 581.479,Z 504.758,A -85,B 0,C 180,E1 -1732.828,E2 -1732.828} C_VEL
LIN {X 0,Y 581.407,Z 520.884,A -85,B 0,C 180,E1 -1733.185,E2 -1733.185} C_VEL
LIN {X 0,Y 581.259,Z 535.636,A -85,B 0,C 180,E1 -1733.658,E2 -1733.658} C_VEL
LIN {X 0,Y 581.127,Z 550.285,A -85,B 0,C 180,E1 -1734.279,E2 -1734.279} C_VEL
LIN {X 0,Y 580.921,Z 564.665,A -85,B 0,C 180,E1 -1735.051,E2 -1735.051} C_VEL
LIN {X 0,Y 580.758,Z 577.652,A -85,B 0,C 180,E1 -1735.909,E2 -1735.909} C_VEL
LIN {X 0,Y 580.601,Z 590.068,A -85,B 0,C 180,E1 -1736.898,E2 -1736.898} C_VEL
LIN {X 0,Y 580.44,Z 601.571,A -85,B 0,C 180,E1 -1737.996,E2 -1737.996} C_VEL
LIN {X 0,Y 580.351,Z 611.653,A -85,B 0,C 180,E1 -1739.143,E2 -1739.143} C_VEL
LIN {X 0,Y 580.241,Z 620.749,A -85,B 0,C 180,E1 -1740.377,E2 -1740.377} C_VEL
LIN {X 0,Y 580.19,Z 628.812,A -85,B 0,C 180,E1 -1741.698,E2 -1741.698} C_VEL
LIN {X 0,Y 580.101,Z 635.473,A -85,B 0,C 180,E1 -1743.037,E2 -1743.037} C_VEL
LIN {X 0,Y 580.085,Z 640.148,A -85,B 0,C 180,E1 -1744.197,E2 -1744.197} C_VEL
LIN {X 0,Y 580.063,Z 644.482,A -85,B 0,C 180,E1 -1745.56,E2 -1745.56} C_VEL
LIN {X 0,Y 580.033,Z 647.56,A -85,B 0,C 180,E1 -1746.898,E2 -1746.898} C_VEL
LIN {X 0,Y 580.016,Z 649.424,A -85,B 0,C 180,E1 -1748.167,E2 -1748.167} C_VEL
LIN {X 0,Y 580.016,Z 650.245,A -85,B 0,C 180,E1 -1749.151,E2 -1749.151} C_VEL
LIN {X 0,Y 580.036,Z 650.462,A -85,B 0,C 180,E1 -1750.24,E2 -1750.24} C_VEL
LIN {X 0,Y 580.05,Z 649.575,A -85,B 0,C 180,E1 -1751.789,E2 -1751.789} C_VEL
LIN {X 0,Y 580.057,Z 648.341,A -85,B 0,C 180,E1 -1752.726,E2 -1752.726} C_VEL
LIN {X 0,Y 580.037,Z 646.553,A -85,B 0,C 180,E1 -1753.68,E2 -1753.68} C_VEL
LIN {X 0,Y 580.09,Z 643.108,A -85,B 0,C 180,E1 -1755.001,E2 -1755.001} C_VEL
LIN {X 0,Y 580.1,Z 638.526,A -85,B 0,C 180,E1 -1756.325,E2 -1756.325} C_VEL
LIN {X 0,Y 580.133,Z 632.728,A -85,B 0,C 180,E1 -1757.644,E2 -1757.644} C_VEL
LIN {X 0,Y 580.18,Z 625.807,A -85,B 0,C 180,E1 -1758.915,E2 -1758.915} C_VEL
LIN {X 0,Y 580.267,Z 616.88,A -85,B 0,C 180,E1 -1760.265,E2 -1760.265} C_VEL
LIN {X 0,Y 580.386,Z 607.691,A -85,B 0,C 180,E1 -1761.418,E2 -1761.418} C_VEL
LIN {X 0,Y 580.472,Z 597.262,A -85,B 0,C 180,E1 -1762.526,E2 -1762.526} C_VEL
LIN {X 0,Y 580.661,Z 584.892,A -85,B 0,C 180,E1 -1763.624,E2 -1763.624} C_VEL
LIN {X 0,Y 580.802,Z 573.198,A -85,B 0,C 180,E1 -1764.491,E2 -1764.491} C_VEL
LIN {X 0,Y 580.979,Z 559.209,A -85,B 0,C 180,E1 -1765.35,E2 -1765.35} C_VEL
LIN {X 0,Y 581.153,Z 545.176,A -85,B 0,C 180,E1 -1766.044,E2 -1766.044} C_VEL
LIN {X 0,Y 581.316,Z 531.167,A -85,B 0,C 180,E1 -1766.587,E2 -1766.587} C_VEL
LIN {X 0,Y 581.421,Z 516.32,A -85,B 0,C 180,E1 -1767.019,E2 -1767.019} C_VEL
LIN {X 0,Y 581.353,Z 504.176,A -85,B 0,C 180,E1 -1767.275,E2 -1767.275} C_VEL
LIN {X 0,Y 580.046,Z 498.364,A -85,B 0,C 180,E1 -1767.424,E2 -1767.424} C_VEL
LIN {X 0,Y 580.047,Z 495.02,A -85,B 0,C 180,E1 -1770.213,E2 -1770.213} C_VEL
LIN {X 0,Y 580.066,Z 492.22,A -85,B 0,C 180,E1 -1772.587,E2 -1772.587} C_VEL
LIN {X 0,Y 580.09,Z 489.057,A -85,B 0,C 180,E1 -1775.318,E2 -1775.318} C_VEL
LIN {X 0,Y 580.062,Z 486.091,A -85,B 0,C 180,E1 -1777.939,E2 -1777.939} C_VEL
LIN {X 0,Y 580.096,Z 483.621,A -85,B 0,C 180,E1 -1780.17,E2 -1780.17} C_VEL
LIN {X 0,Y 580.223,Z 481.111,A -85,B 0,C 180,E1 -1783.113,E2 -1783.113} C_VEL
LIN {X 0,Y 580.188,Z 478.201,A -85,B 0,C 180,E1 -1785.979,E2 -1785.979} C_VEL
LIN {X 0,Y 580.179,Z 476.845,A -85,B 0,C 180,E1 -1787.406,E2 -1787.406} C_VEL
LIN {X 0,Y 580.303,Z 476.822,A -85,B 0,C 180,E1 -1789.533,E2 -1789.533} C_VEL
LIN {X 0,Y 580.327,Z 476.822,A -85,B 0,C 180,E1 -1792.344,E2 -1792.344} C_VEL
LIN {X 0,Y 580.338,Z 476.817,A -85,B 0,C 180,E1 -1795.137,E2 -1795.137} C_VEL
LIN {X 0,Y 580.337,Z 476.822,A -85,B 0,C 180,E1 -1797.918,E2 -1797.918} C_VEL
LIN {X 0,Y 580.361,Z 476.813,A -85,B 0,C 180,E1 -1800.694,E2 -1800.694} C_VEL
LIN {X 0,Y 580.281,Z 476.832,A -85,B 0,C 180,E1 -1803.472,E2 -1803.472} C_VEL
LIN {X 0,Y 580.325,Z 476.823,A -85,B 0,C 180,E1 -1805.559,E2 -1805.559} C_VEL
LIN {X 0,Y 580.331,Z 476.817,A -85,B 0,C 180,E1 -1808.356,E2 -1808.356} C_VEL
LIN {X 0,Y 580.329,Z 476.823,A -85,B 0,C 180,E1 -1811.208,E2 -1811.208} C_VEL
LIN {X 0,Y 580.31,Z 476.822,A -85,B 0,C 180,E1 -1814.339,E2 -1814.339} C_VEL
LIN {X 0,Y 580.307,Z 476.826,A -85,B 0,C 180,E1 -1816.914,E2 -1816.914} C_VEL
LIN {X 0,Y 580.302,Z 476.821,A -85,B 0,C 180,E1 -1819.822,E2 -1819.822} C_VEL
LIN {X 0,Y 580.27,Z 476.828,A -85,B 0,C 180,E1 -1822.053,E2 -1822.053} C_VEL
LIN {X 0,Y 580.305,Z 476.82,A -85,B 0,C 180,E1 -1825.08,E2 -1825.08} C_VEL
LIN {X 0,Y 580.317,Z 476.824,A -85,B 0,C 180,E1 -1827.863,E2 -1827.863} C_VEL
LIN {X 0,Y 580.295,Z 476.822,A -85,B 0,C 180,E1 -1830.697,E2 -1830.697} C_VEL
LIN {X 0,Y 580.301,Z 476.823,A -85,B 0,C 180,E1 -1833.317,E2 -1833.317} C_VEL
LIN {X 0,Y 580.323,Z 476.826,A -85,B 0,C 180,E1 -1835.768,E2 -1835.768} C_VEL
LIN {X 0,Y 580.285,Z 476.824,A -85,B 0,C 180,E1 -1838.146,E2 -1838.146} C_VEL
LIN {X 0,Y 580.298,Z 476.823,A -85,B 0,C 180,E1 -1840.843,E2 -1840.843} C_VEL
LIN {X 0,Y 580.285,Z 476.828,A -85,B 0,C 180,E1 -1843.657,E2 -1843.657} C_VEL
LIN {X 0,Y 580.29,Z 476.828,A -85,B 0,C 180,E1 -1846.608,E2 -1846.608} C_VEL
LIN {X 0,Y 580.333,Z 476.874,A -85,B 0,C 180,E1 -1847.493,E2 -1847.493} C_VEL
LIN {X 0,Y 580.749,Z 481.153,A -85,B 0,C 180,E1 -1849.195,E2 -1849.195} C_VEL
LIN {X 0,Y 580.678,Z 487.321,A -85,B 0,C 180,E1 -1851.442,E2 -1851.442} C_VEL
LIN {X 0,Y 580.603,Z 495.205,A -85,B 0,C 180,E1 -1854.195,E2 -1854.195} C_VEL
LIN {X 0,Y 580.545,Z 502.698,A -85,B 0,C 180,E1 -1856.647,E2 -1856.647} C_VEL
LIN {X 0,Y 580.551,Z 511.587,A -85,B 0,C 180,E1 -1859.44,E2 -1859.44} C_VEL
LIN {X 0,Y 580.488,Z 519.9,A -85,B 0,C 180,E1 -1862.106,E2 -1862.106} C_VEL
LIN {X 0,Y 580.407,Z 527.679,A -85,B 0,C 180,E1 -1864.541,E2 -1864.541} C_VEL
LIN {X 0,Y 580.332,Z 536.343,A -85,B 0,C 180,E1 -1867.199,E2 -1867.199} C_VEL
LIN {X 0,Y 580.272,Z 545.008,A -85,B 0,C 180,E1 -1869.807,E2 -1869.807} C_VEL
LIN {X 0,Y 580.234,Z 554.414,A -85,B 0,C 180,E1 -1872.592,E2 -1872.592} C_VEL
LIN {X 0,Y 581.48,Z 560.045,A -85,B 0,C 180,E1 -1872.712,E2 -1872.712} C_VEL
LIN {X 0,Y 581.417,Z 575.475,A -85,B 0,C 180,E1 -1873.005,E2 -1873.005} C_VEL
LIN {X 0,Y 581.314,Z 590.91,A -85,B 0,C 180,E1 -1873.449,E2 -1873.449} C_VEL
LIN {X 0,Y 581.199,Z 603.836,A -85,B 0,C 180,E1 -1873.942,E2 -1873.942} C_VEL
LIN {X 0,Y 581.004,Z 618.523,A -85,B 0,C 180,E1 -1874.656,E2 -1874.656} C_VEL
LIN {X 0,Y 580.834,Z 631.873,A -85,B 0,C 180,E1 -1875.463,E2 -1875.463} C_VEL
LIN {X 0,Y 580.677,Z 644.013,A -85,B 0,C 180,E1 -1876.349,E2 -1876.349} C_VEL
LIN {X 0,Y 580.541,Z 656.189,A -85,B 0,C 180,E1 -1877.414,E2 -1877.414} C_VEL
LIN {X 0,Y 580.385,Z 666.704,A -85,B 0,C 180,E1 -1878.51,E2 -1878.51} C_VEL
LIN {X 0,Y 580.308,Z 676.369,A -85,B 0,C 180,E1 -1879.71,E2 -1879.71} C_VEL
LIN {X 0,Y 580.208,Z 684.651,A -85,B 0,C 180,E1 -1880.94,E2 -1880.94} C_VEL
LIN {X 0,Y 580.165,Z 692.424,A -85,B 0,C 180,E1 -1882.342,E2 -1882.342} C_VEL
LIN {X 0,Y 580.092,Z 698.606,A -85,B 0,C 180,E1 -1883.74,E2 -1883.74} C_VEL
LIN {X 0,Y 580.041,Z 703.383,A -85,B 0,C 180,E1 -1885.134,E2 -1885.134} C_VEL
LIN {X 0,Y 580.105,Z 706.887,A -85,B 0,C 180,E1 -1886.527,E2 -1886.527} C_VEL
LIN {X 0,Y 580.036,Z 709.193,A -85,B 0,C 180,E1 -1887.917,E2 -1887.917} C_VEL
LIN {X 0,Y 580.038,Z 710.35,A -85,B 0,C 180,E1 -1889.305,E2 -1889.305} C_VEL
LIN {X 0,Y 580.038,Z 710.35,A -85,B 0,C 180,E1 -1890.694,E2 -1890.694} C_VEL
LIN {X 0,Y 580.036,Z 709.193,A -85,B 0,C 180,E1 -1892.083,E2 -1892.083} C_VEL
LIN {X 0,Y 580.105,Z 706.887,A -85,B 0,C 180,E1 -1893.472,E2 -1893.472} C_VEL
LIN {X 0,Y 580.041,Z 703.386,A -85,B 0,C 180,E1 -1894.865,E2 -1894.865} C_VEL
LIN {X 0,Y 580.091,Z 698.61,A -85,B 0,C 180,E1 -1896.259,E2 -1896.259} C_VEL
LIN {X 0,Y 580.168,Z 692.427,A -85,B 0,C 180,E1 -1897.657,E2 -1897.657} C_VEL
LIN {X 0,Y 580.207,Z 684.654,A -85,B 0,C 180,E1 -1899.059,E2 -1899.059} C_VEL
LIN {X 0,Y 580.308,Z 676.374,A -85,B 0,C 180,E1 -1900.29,E2 -1900.29} C_VEL
LIN {X 0,Y 580.382,Z 666.4,A -85,B 0,C 180,E1 -1901.525,E2 -1901.525} C_VEL
LIN {X 0,Y 580.54,Z 656.197,A -85,B 0,C 180,E1 -1902.586,E2 -1902.586} C_VEL
LIN {X 0,Y 580.677,Z 644.025,A -85,B 0,C 180,E1 -1903.651,E2 -1903.651} C_VEL
LIN {X 0,Y 580.844,Z 631.816,A -85,B 0,C 180,E1 -1904.541,E2 -1904.541} C_VEL
LIN {X 0,Y 581.003,Z 618.533,A -85,B 0,C 180,E1 -1905.343,E2 -1905.343} C_VEL
LIN {X 0,Y 581.201,Z 603.852,A -85,B 0,C 180,E1 -1906.057,E2 -1906.057} C_VEL
LIN {X 0,Y 581.339,Z 589.636,A -85,B 0,C 180,E1 -1906.595,E2 -1906.595} C_VEL
LIN {X 0,Y 581.428,Z 574.643,A -85,B 0,C 180,E1 -1907.015,E2 -1907.015} C_VEL
LIN {X 0,Y 581.378,Z 559.674,A -85,B 0,C 180,E1 -1907.297,E2 -1907.297} C_VEL
LIN {X 0,Y 580.213,Z 554.394,A -85,B 0,C 180,E1 -1907.415,E2 -1907.415} C_VEL
LIN {X 0,Y 580.271,Z 545.01,A -85,B 0,C 180,E1 -1910.192,E2 -1910.192} C_VEL
LIN {X 0,Y 580.326,Z 535.634,A -85,B 0,C 180,E1 -1913.017,E2 -1913.017} C_VEL
LIN {X 0,Y 580.426,Z 526.443,A -85,B 0,C 180,E1 -1915.842,E2 -1915.842} C_VEL
LIN {X 0,Y 580.495,Z 517.779,A -85,B 0,C 180,E1 -1918.568,E2 -1918.568} C_VEL
LIN {X 0,Y 580.585,Z 509.1,A -85,B 0,C 180,E1 -1921.366,E2 -1921.366} C_VEL
LIN {X 0,Y 580.618,Z 500.249,A -85,B 0,C 180,E1 -1924.216,E2 -1924.216} C_VEL
LIN {X 0,Y 580.65,Z 492.017,A -85,B 0,C 180,E1 -1926.98,E2 -1926.98} C_VEL
LIN {X 0,Y 580.77,Z 485.661,A -85,B 0,C 180,E1 -1929.243,E2 -1929.243} C_VEL
LIN {X 0,Y 580.774,Z 479.882,A -85,B 0,C 180,E1 -1931.387,E2 -1931.387} C_VEL
LIN {X 0,Y 580.308,Z 476.828,A -85,B 0,C 180,E1 -1932.606,E2 -1932.606} C_VEL
LIN {X 0,Y 580.267,Z 476.833,A -85,B 0,C 180,E1 -1935.608,E2 -1935.608} C_VEL
LIN {X 0,Y 580.313,Z 476.825,A -85,B 0,C 180,E1 -1938.234,E2 -1938.234} C_VEL
LIN {X 0,Y 580.289,Z 476.831,A -85,B 0,C 180,E1 -1940.966,E2 -1940.966} C_VEL
LIN {X 0,Y 580.289,Z 476.828,A -85,B 0,C 180,E1 -1943.598,E2 -1943.598} C_VEL
LIN {X 0,Y 580.315,Z 476.826,A -85,B 0,C 180,E1 -1946.145,E2 -1946.145} C_VEL
LIN {X 0,Y 580.285,Z 476.831,A -85,B 0,C 180,E1 -1948.615,E2 -1948.615} C_VEL
LIN {X 0,Y 580.291,Z 476.83,A -85,B 0,C 180,E1 -1951.024,E2 -1951.024} C_VEL
LIN {X 0,Y 580.321,Z 476.824,A -85,B 0,C 180,E1 -1953.657,E2 -1953.657} C_VEL
LIN {X 0,Y 580.271,Z 476.833,A -85,B 0,C 180,E1 -1956.442,E2 -1956.442} C_VEL
LIN {X 0,Y 580.277,Z 476.831,A -85,B 0,C 180,E1 -1959.438,E2 -1959.438} C_VEL
LIN {X 0,Y 580.277,Z 476.831,A -85,B 0,C 180,E1 -1961.646,E2 -1961.646} C_VEL
LIN {X 0,Y 580.277,Z 476.831,A -85,B 0,C 180,E1 -1963.826,E2 -1963.826} C_VEL
LIN {X 0,Y 580.271,Z 476.83,A -85,B 0,C 180,E1 -1966.696,E2 -1966.696} C_VEL
LIN {X 0,Y 580.298,Z 476.83,A -85,B 0,C 180,E1 -1969.533,E2 -1969.533} C_VEL
LIN {X 0,Y 580.333,Z 476.822,A -85,B 0,C 180,E1 -1972.345,E2 -1972.345} C_VEL
LIN {X 0,Y 580.336,Z 476.825,A -85,B 0,C 180,E1 -1975.137,E2 -1975.137} C_VEL
LIN {X 0,Y 580.332,Z 476.823,A -85,B 0,C 180,E1 -1977.918,E2 -1977.918} C_VEL
LIN {X 0,Y 580.36,Z 476.821,A -85,B 0,C 180,E1 -1980.694,E2 -1980.694} C_VEL
LIN {X 0,Y 580.287,Z 476.829,A -85,B 0,C 180,E1 -1983.472,E2 -1983.472} C_VEL
LIN {X 0,Y 580.331,Z 476.823,A -85,B 0,C 180,E1 -1985.56,E2 -1985.56} C_VEL
LIN {X 0,Y 580.329,Z 476.825,A -85,B 0,C 180,E1 -1988.356,E2 -1988.356} C_VEL
LIN {X 0,Y 580.323,Z 476.824,A -85,B 0,C 180,E1 -1991.209,E2 -1991.209} C_VEL
LIN {X 0,Y 580.306,Z 476.826,A -85,B 0,C 180,E1 -1994.34,E2 -1994.34} C_VEL
LIN {X 0,Y 580.306,Z 476.827,A -85,B 0,C 180,E1 -1996.916,E2 -1996.916} C_VEL
LIN {X 0,Y 580.302,Z 476.827,A -85,B 0,C 180,E1 -1999.823,E2 -1999.823} C_VEL
LIN {X 0,Y 580.279,Z 476.83,A -85,B 0,C 180,E1 -2001.346,E2 -2001.346} C_VEL
LIN {X 0,Y 579.582,Z 476.917,A -85,B 0,C 180,E1 -2001.925,E2 -2001.925} C_VEL
LIN {X 0,Y 576.704,Z 477.276,A -85,B 0,C 180,E1 -2002.865,E2 -2002.865} C_VEL
LIN {X 0,Y 574.309,Z 477.576,A -85,B 0,C 180,E1 -2003.621,E2 -2003.621} C_VEL
LIN {X 0,Y 573.31,Z 477.697,A -85,B 0,C 180,E1 -2004.205,E2 -2004.205} C_VEL
LIN {X 0,Y 573.244,Z 477.706,A -85,B 0,C 180,E1 -2004.402,E2 -2004.402} C_VEL
LIN {X 0,Y 573.264,Z 477.705,A -85,B 0,C 180,E1 -2006.976,E2 -2006.976} C_VEL
LIN {X 0,Y 573.249,Z 477.706,A -85,B 0,C 180,E1 -2009.491,E2 -2009.491} C_VEL
LIN {X 0,Y 573.252,Z 477.706,A -85,B 0,C 180,E1 -2012.23,E2 -2012.23} C_VEL
LIN {X 0,Y 573.248,Z 477.708,A -85,B 0,C 180,E1 -2014.775,E2 -2014.775} C_VEL
LIN {X 0,Y 573.25,Z 477.706,A -85,B 0,C 180,E1 -2017.167,E2 -2017.167} C_VEL
LIN {X 0,Y 573.248,Z 477.706,A -85,B 0,C 180,E1 -2019.608,E2 -2019.608} C_VEL
LIN {X 0,Y 573.238,Z 477.709,A -85,B 0,C 180,E1 -2022.401,E2 -2022.401} C_VEL
LIN {X 0,Y 573.223,Z 477.71,A -85,B 0,C 180,E1 -2024.676,E2 -2024.676} C_VEL
LIN {X 0,Y 573.241,Z 477.706,A -85,B 0,C 180,E1 -2027.359,E2 -2027.359} C_VEL
LIN {X 0,Y 573.272,Z 477.703,A -85,B 0,C 180,E1 -2029.479,E2 -2029.479} C_VEL
LIN {X 0,Y 573.238,Z 477.709,A -85,B 0,C 180,E1 -2032.194,E2 -2032.194} C_VEL
LIN {X 0,Y 573.254,Z 477.705,A -85,B 0,C 180,E1 -2034.817,E2 -2034.817} C_VEL
LIN {X 0,Y 573.255,Z 477.704,A -85,B 0,C 180,E1 -2037.356,E2 -2037.356} C_VEL
LIN {X 0,Y 573.251,Z 477.706,A -85,B 0,C 180,E1 -2039.825,E2 -2039.825} C_VEL
LIN {X 0,Y 573.291,Z 477.702,A -85,B 0,C 180,E1 -2042.236,E2 -2042.236} C_VEL
LIN {X 0,Y 573.272,Z 477.702,A -85,B 0,C 180,E1 -2045.122,E2 -2045.122} C_VEL
LIN {X 0,Y 573.239,Z 477.709,A -85,B 0,C 180,E1 -2047.663,E2 -2047.663} C_VEL
LIN {X 0,Y 573.269,Z 477.702,A -85,B 0,C 180,E1 -2050.671,E2 -2050.671} C_VEL
LIN {X 0,Y 573.256,Z 477.705,A -85,B 0,C 180,E1 -2053.623,E2 -2053.623} C_VEL
LIN {X 0,Y 573.278,Z 477.702,A -85,B 0,C 180,E1 -2055.808,E2 -2055.808} C_VEL
LIN {X 0,Y 573.268,Z 477.705,A -85,B 0,C 180,E1 -2058.746,E2 -2058.746} C_VEL
LIN {X 0,Y 573.259,Z 477.704,A -85,B 0,C 180,E1 -2061.541,E2 -2061.541} C_VEL
LIN {X 0,Y 573.251,Z 477.705,A -85,B 0,C 180,E1 -2063.666,E2 -2063.666} C_VEL
LIN {X 0,Y 573.236,Z 477.707,A -85,B 0,C 180,E1 -2065.782,E2 -2065.782} C_VEL
LIN {X 0,Y 573.316,Z 477.697,A -85,B 0,C 180,E1 -2067.893,E2 -2067.893} C_VEL
LIN {X 0,Y 573.337,Z 477.695,A -85,B 0,C 180,E1 -2070.703,E2 -2070.703} C_VEL
LIN {X 0,Y 573.121,Z 477.724,A -85,B 0,C 180,E1 -2072.812,E2 -2072.812} C_VEL
LIN {X 0,Y 573.077,Z 477.934,A -85,B 0,C 180,E1 -2073.516,E2 -2073.516} C_VEL
LIN {X 0,Y 573.077,Z 480.011,A -85,B 0,C 180,E1 -2075.631,E2 -2075.631} C_VEL
LIN {X 0,Y 573.076,Z 482.802,A -85,B 0,C 180,E1 -2078.463,E2 -2078.463} C_VEL
LIN {X 0,Y 573.039,Z 485.582,A -85,B 0,C 180,E1 -2081.317,E2 -2081.317} C_VEL
LIN {X 0,Y 573.047,Z 488.934,A -85,B 0,C 180,E1 -2084.33,E2 -2084.33} C_VEL
LIN {X 0,Y 572.978,Z 492.118,A -85,B 0,C 180,E1 -2087.12,E2 -2087.12} C_VEL
LIN {X 0,Y 572.975,Z 495.572,A -85,B 0,C 180,E1 -2090.087,E2 -2090.087} C_VEL
LIN {X 0,Y 572.964,Z 498.47,A -85,B 0,C 180,E1 -2092.468,E2 -2092.468} C_VEL
LIN {X 0,Y 574.681,Z 505.638,A -85,B 0,C 180,E1 -2092.634,E2 -2092.634} C_VEL
LIN {X 0,Y 574.615,Z 521.328,A -85,B 0,C 180,E1 -2092.993,E2 -2092.993} C_VEL
LIN {X 0,Y 574.41,Z 536.515,A -85,B 0,C 180,E1 -2093.491,E2 -2093.491} C_VEL
LIN {X 0,Y 574.262,Z 550.729,A -85,B 0,C 180,E1 -2094.108,E2 -2094.108} C_VEL
LIN {X 0,Y 574.013,Z 564.246,A -85,B 0,C 180,E1 -2094.841,E2 -2094.841} C_VEL
LIN {X 0,Y 573.821,Z 578.152,A -85,B 0,C 180,E1 -2095.772,E2 -2095.772} C_VEL
LIN {X 0,Y 573.621,Z 589.956,A -85,B 0,C 180,E1 -2096.726,E2 -2096.726} C_VEL
LIN {X 0,Y 573.444,Z 600.701,A -85,B 0,C 180,E1 -2097.757,E2 -2097.757} C_VEL
LIN {X 0,Y 573.296,Z 611.284,A -85,B 0,C 180,E1 -2098.962,E2 -2098.962} C_VEL
LIN {X 0,Y 573.203,Z 620.209,A -85,B 0,C 180,E1 -2100.178,E2 -2100.178} C_VEL
LIN {X 0,Y 573.102,Z 627.776,A -85,B 0,C 180,E1 -2101.411,E2 -2101.411} C_VEL
LIN {X 0,Y 573.033,Z 634.146,A -85,B 0,C 180,E1 -2102.659,E2 -2102.659} C_VEL
LIN {X 0,Y 573.022,Z 639.432,A -85,B 0,C 180,E1 -2103.921,E2 -2103.921} C_VEL
LIN {X 0,Y 572.963,Z 643.641,A -85,B 0,C 180,E1 -2105.205,E2 -2105.205} C_VEL
LIN {X 0,Y 572.936,Z 645.911,A -85,B 0,C 180,E1 -2106.071,E2 -2106.071} C_VEL
LIN {X 0,Y 572.927,Z 648.01,A -85,B 0,C 180,E1 -2107.122,E2 -2107.122} C_VEL
LIN {X 0,Y 572.928,Z 649.566,A -85,B 0,C 180,E1 -2108.272,E2 -2108.272} C_VEL
LIN {X 0,Y 572.922,Z 650.415,A -85,B 0,C 180,E1 -2109.634,E2 -2109.634} C_VEL
LIN {X 0,Y 572.937,Z 650.394,A -85,B 0,C 180,E1 -2110.551,E2 -2110.551} C_VEL
LIN {X 0,Y 572.964,Z 649.835,A -85,B 0,C 180,E1 -2111.562,E2 -2111.562} C_VEL
LIN {X 0,Y 572.959,Z 648.575,A -85,B 0,C 180,E1 -2112.61,E2 -2112.61} C_VEL
LIN {X 0,Y 572.937,Z 646.736,A -85,B 0,C 180,E1 -2113.636,E2 -2113.636} C_VEL
LIN {X 0,Y 572.994,Z 643.372,A -85,B 0,C 180,E1 -2114.975,E2 -2114.975} C_VEL
LIN {X 0,Y 573.008,Z 638.716,A -85,B 0,C 180,E1 -2116.355,E2 -2116.355} C_VEL
LIN {X 0,Y 573.056,Z 633.457,A -85,B 0,C 180,E1 -2117.582,E2 -2117.582} C_VEL
LIN {X 0,Y 573.102,Z 625.96,A -85,B 0,C 180,E1 -2118.998,E2 -2118.998} C_VEL
LIN {X 0,Y 573.244,Z 616.875,A -85,B 0,C 180,E1 -2120.392,E2 -2120.392} C_VEL
LIN {X 0,Y 573.401,Z 606.79,A -85,B 0,C 180,E1 -2121.667,E2 -2121.667} C_VEL
LIN {X 0,Y 573.509,Z 596.073,A -85,B 0,C 180,E1 -2122.8,E2 -2122.8} C_VEL
LIN {X 0,Y 573.736,Z 583.715,A -85,B 0,C 180,E1 -2123.888,E2 -2123.888} C_VEL
LIN {X 0,Y 573.913,Z 570.369,A -85,B 0,C 180,E1 -2124.861,E2 -2124.861} C_VEL
LIN {X 0,Y 574.126,Z 557.535,A -85,B 0,C 180,E1 -2125.633,E2 -2125.633} C_VEL
LIN {X 0,Y 574.332,Z 543.524,A -85,B 0,C 180,E1 -2126.314,E2 -2126.314} C_VEL
LIN {X 0,Y 574.512,Z 529.101,A -85,B 0,C 180,E1 -2126.861,E2 -2126.861} C_VEL
LIN {X 0,Y 574.664,Z 513.768,A -85,B 0,C 180,E1 -2127.288,E2 -2127.288} C_VEL
LIN {X 0,Y 574.623,Z 505.51,A -85,B 0,C 180,E1 -2127.46,E2 -2127.46} C_VEL
LIN {X 0,Y 572.949,Z 498.383,A -85,B 0,C 180,E1 -2127.63,E2 -2127.63} C_VEL
LIN {X 0,Y 572.982,Z 494.85,A -85,B 0,C 180,E1 -2130.618,E2 -2130.618} C_VEL
LIN {X 0,Y 573.004,Z 491.446,A -85,B 0,C 180,E1 -2133.553,E2 -2133.553} C_VEL
LIN {X 0,Y 573.002,Z 488.527,A -85,B 0,C 180,E1 -2136.124,E2 -2136.124} C_VEL
LIN {X 0,Y 573.015,Z 485.212,A -85,B 0,C 180,E1 -2139.164,E2 -2139.164} C_VEL
LIN {X 0,Y 573.075,Z 483.307,A -85,B 0,C 180,E1 -2141.406,E2 -2141.406} C_VEL
LIN {X 0,Y 573.126,Z 481.242,A -85,B 0,C 180,E1 -2143.618,E2 -2143.618} C_VEL
LIN {X 0,Y 573.119,Z 478.363,A -85,B 0,C 180,E1 -2146.526,E2 -2146.526} C_VEL
LIN {X 0,Y 573.122,Z 477.724,A -85,B 0,C 180,E1 -2147.248,E2 -2147.248} C_VEL
LIN {X 0,Y 573.268,Z 477.698,A -85,B 0,C 180,E1 -2149.403,E2 -2149.403} C_VEL
LIN {X 0,Y 573.278,Z 477.701,A -85,B 0,C 180,E1 -2152.25,E2 -2152.25} C_VEL
LIN {X 0,Y 573.31,Z 477.692,A -85,B 0,C 180,E1 -2155.077,E2 -2155.077} C_VEL
LIN {X 0,Y 573.307,Z 477.698,A -85,B 0,C 180,E1 -2157.892,E2 -2157.892} C_VEL
LIN {X 0,Y 573.331,Z 477.689,A -85,B 0,C 180,E1 -2160.702,E2 -2160.702} C_VEL
LIN {X 0,Y 573.233,Z 477.709,A -85,B 0,C 180,E1 -2163.514,E2 -2163.514} C_VEL
LIN {X 0,Y 573.291,Z 477.698,A -85,B 0,C 180,E1 -2165.628,E2 -2165.628} C_VEL
LIN {X 0,Y 573.287,Z 477.695,A -85,B 0,C 180,E1 -2168.459,E2 -2168.459} C_VEL
LIN {X 0,Y 573.295,Z 477.698,A -85,B 0,C 180,E1 -2171.311,E2 -2171.311} C_VEL
LIN {X 0,Y 573.276,Z 477.699,A -85,B 0,C 180,E1 -2174.424,E2 -2174.424} C_VEL
LIN {X 0,Y 573.253,Z 477.701,A -85,B 0,C 180,E1 -2177.112,E2 -2177.112} C_VEL
LIN {X 0,Y 573.252,Z 477.701,A -85,B 0,C 180,E1 -2180.076,E2 -2180.076} C_VEL
LIN {X 0,Y 573.234,Z 477.709,A -85,B 0,C 180,E1 -2182.338,E2 -2182.338} C_VEL
LIN {X 0,Y 573.254,Z 477.699,A -85,B 0,C 180,E1 -2185.41,E2 -2185.41} C_VEL
LIN {X 0,Y 573.261,Z 477.706,A -85,B 0,C 180,E1 -2188.032,E2 -2188.032} C_VEL
LIN {X 0,Y 573.24,Z 477.701,A -85,B 0,C 180,E1 -2190.885,E2 -2190.885} C_VEL
LIN {X 0,Y 573.258,Z 477.703,A -85,B 0,C 180,E1 -2193.524,E2 -2193.524} C_VEL
LIN {X 0,Y 573.258,Z 477.703,A -85,B 0,C 180,E1 -2196.048,E2 -2196.048} C_VEL
LIN {X 0,Y 573.246,Z 477.699,A -85,B 0,C 180,E1 -2198.701,E2 -2198.701} C_VEL
LIN {X 0,Y 573.251,Z 477.706,A -85,B 0,C 180,E1 -2201.596,E2 -2201.596} C_VEL
LIN {X 0,Y 573.237,Z 477.703,A -85,B 0,C 180,E1 -2204.333,E2 -2204.333} C_VEL
LIN {X 0,Y 573.274,Z 477.739,A -85,B 0,C 180,E1 -2207.22,E2 -2207.22} C_VEL
LIN {X 0,Y 573.788,Z 482.181,A -85,B 0,C 180,E1 -2209.041,E2 -2209.041} C_VEL
LIN {X 0,Y 573.68,Z 489.215,A -85,B 0,C 180,E1 -2211.632,E2 -2211.632} C_VEL
LIN {X 0,Y 573.632,Z 497.121,A -85,B 0,C 180,E1 -2214.412,E2 -2214.412} C_VEL
LIN {X 0,Y 573.529,Z 504.806,A -85,B 0,C 180,E1 -2216.955,E2 -2216.955} C_VEL
LIN {X 0,Y 573.547,Z 512.785,A -85,B 0,C 180,E1 -2219.451,E2 -2219.451} C_VEL
LIN {X 0,Y 573.449,Z 521.49,A -85,B 0,C 180,E1 -2222.244,E2 -2222.244} C_VEL
LIN {X 0,Y 573.384,Z 528.916,A -85,B 0,C 180,E1 -2224.596,E2 -2224.596} C_VEL
LIN {X 0,Y 573.287,Z 537.581,A -85,B 0,C 180,E1 -2227.284,E2 -2227.284} C_VEL
LIN {X 0,Y 573.221,Z 546.245,A -85,B 0,C 180,E1 -2229.922,E2 -2229.922} C_VEL
LIN {X 0,Y 573.166,Z 554.425,A -85,B 0,C 180,E1 -2232.373,E2 -2232.373} C_VEL
LIN {X 0,Y 574.726,Z 561.118,A -85,B 0,C 180,E1 -2232.519,E2 -2232.519} C_VEL
LIN {X 0,Y 574.632,Z 576.932,A -85,B 0,C 180,E1 -2232.835,E2 -2232.835} C_VEL
LIN {X 0,Y 574.493,Z 592.205,A -85,B 0,C 180,E1 -2233.293,E2 -2233.293} C_VEL
LIN {X 0,Y 574.349,Z 605.822,A -85,B 0,C 180,E1 -2233.836,E2 -2233.836} C_VEL
LIN {X 0,Y 574.099,Z 620.102,A -85,B 0,C 180,E1 -2234.558,E2 -2234.558} C_VEL
LIN {X 0,Y 573.888,Z 633.699,A -85,B 0,C 180,E1 -2235.411,E2 -2235.411} C_VEL
LIN {X 0,Y 573.689,Z 646.163,A -85,B 0,C 180,E1 -2236.36,E2 -2236.36} C_VEL
LIN {X 0,Y 573.511,Z 657.971,A -85,B 0,C 180,E1 -2237.437,E2 -2237.437} C_VEL
LIN {X 0,Y 573.349,Z 667.9,A -85,B 0,C 180,E1 -2238.51,E2 -2238.51} C_VEL
LIN {X 0,Y 573.256,Z 677.618,A -85,B 0,C 180,E1 -2239.76,E2 -2239.76} C_VEL
LIN {X 0,Y 573.136,Z 685.72,A -85,B 0,C 180,E1 -2241.005,E2 -2241.005} C_VEL
LIN {X 0,Y 573.094,Z 692.424,A -85,B 0,C 180,E1 -2242.247,E2 -2242.247} C_VEL
LIN {X 0,Y 573.013,Z 698.606,A -85,B 0,C 180,E1 -2243.662,E2 -2243.662} C_VEL
LIN {X 0,Y 572.951,Z 703.384,A -85,B 0,C 180,E1 -2245.074,E2 -2245.074} C_VEL
LIN {X 0,Y 573.004,Z 706.888,A -85,B 0,C 180,E1 -2246.484,E2 -2246.484} C_VEL
LIN {X 0,Y 572.935,Z 709.192,A -85,B 0,C 180,E1 -2247.891,E2 -2247.891} C_VEL
LIN {X 0,Y 572.938,Z 710.349,A -85,B 0,C 180,E1 -2249.297,E2 -2249.297} C_VEL
LIN {X 0,Y 572.938,Z 710.349,A -85,B 0,C 180,E1 -2250.702,E2 -2250.702} C_VEL
LIN {X 0,Y 572.935,Z 709.192,A -85,B 0,C 180,E1 -2252.109,E2 -2252.109} C_VEL
LIN {X 0,Y 573.004,Z 706.887,A -85,B 0,C 180,E1 -2253.515,E2 -2253.515} C_VEL
LIN {X 0,Y 572.951,Z 703.386,A -85,B 0,C 180,E1 -2254.925,E2 -2254.925} C_VEL
LIN {X 0,Y 573.012,Z 698.61,A -85,B 0,C 180,E1 -2256.337,E2 -2256.337} C_VEL
LIN {X 0,Y 573.095,Z 692.426,A -85,B 0,C 180,E1 -2257.752,E2 -2257.752} C_VEL
LIN {X 0,Y 573.136,Z 684.653,A -85,B 0,C 180,E1 -2259.172,E2 -2259.172} C_VEL
LIN {X 0,Y 573.27,Z 676.373,A -85,B 0,C 180,E1 -2260.417,E2 -2260.417} C_VEL
LIN {X 0,Y 573.384,Z 666.397,A -85,B 0,C 180,E1 -2261.667,E2 -2261.667} C_VEL
LIN {X 0,Y 573.567,Z 656.196,A -85,B 0,C 180,E1 -2262.741,E2 -2262.741} C_VEL
LIN {X 0,Y 573.742,Z 644.026,A -85,B 0,C 180,E1 -2263.819,E2 -2263.819} C_VEL
LIN {X 0,Y 573.96,Z 630.91,A -85,B 0,C 180,E1 -2264.78,E2 -2264.78} C_VEL
LIN {X 0,Y 574.138,Z 616.88,A -85,B 0,C 180,E1 -2265.622,E2 -2265.622} C_VEL
LIN {X 0,Y 574.358,Z 602.813,A -85,B 0,C 180,E1 -2266.299,E2 -2266.299} C_VEL
LIN {X 0,Y 574.524,Z 588.324,A -85,B 0,C 180,E1 -2266.843,E2 -2266.843} C_VEL
LIN {X 0,Y 574.708,Z 572.903,A -85,B 0,C 180,E1 -2267.263,E2 -2267.263} C_VEL
LIN {X 0,Y 574.603,Z 560.766,A -85,B 0,C 180,E1 -2267.491,E2 -2267.491} C_VEL
LIN {X 0,Y 573.17,Z 554.372,A -85,B 0,C 180,E1 -2267.642,E2 -2267.642} C_VEL
LIN {X 0,Y 573.229,Z 545.01,A -85,B 0,C 180,E1 -2270.451,E2 -2270.451} C_VEL
LIN {X 0,Y 573.341,Z 535.109,A -85,B 0,C 180,E1 -2273.476,E2 -2273.476} C_VEL
LIN {X 0,Y 573.464,Z 525.31,A -85,B 0,C 180,E1 -2276.538,E2 -2276.538} C_VEL
LIN {X 0,Y 573.532,Z 515.962,A -85,B 0,C 180,E1 -2279.539,E2 -2279.539} C_VEL
LIN {X 0,Y 573.596,Z 507.432,A -85,B 0,C 180,E1 -2282.283,E2 -2282.283} C_VEL
LIN {X 0,Y 573.614,Z 499.693,A -85,B 0,C 180,E1 -2284.826,E2 -2284.826} C_VEL
